LIN {X 0,Y 270.125,Z 311.646,A -85,B 0,C 180,E1 -17954.625,E2 -17954.625} C_VEL
LIN {X 0,Y 270.147,Z 311.642,A -85,B 0,C 180,E1 -17957.437,E2 -17957.437} C_VEL
LIN {X 0,Y 270.147,Z 311.617,A -85,B 0,C 180,E1 -17961.364,E2 -17961.364} C_VEL
LIN {X 0,Y 270.193,Z 311.638,A -85,B 0,C 180,E1 -17965.093,E2 -17965.093} C_VEL
LIN {X 0,Y 270.18,Z 311.636,A -85,B 0,C 180,E1 -17969.136,E2 -17969.136} C_VEL
LIN {X 0,Y 270.194,Z 311.636,A -85,B 0,C 180,E1 -17972.172,E2 -17972.172} C_VEL
LIN {X 0,Y 270.176,Z 311.639,A -85,B 0,C 180,E1 -17975.564,E2 -17975.564} C_VEL
LIN {X 0,Y 270.213,Z 311.635,A -85,B 0,C 180,E1 -17980.238,E2 -17980.238} C_VEL
LIN {X 0,Y 270.332,Z 311.614,A -85,B 0,C 180,E1 -17984.931,E2 -17984.931} C_VEL
LIN {X 0,Y 270.379,Z 311.614,A -85,B 0,C 180,E1 -17989.516,E2 -17989.516} C_VEL
LIN {X 0,Y 270.555,Z 311.591,A -85,B 0,C 180,E1 -17992.537,E2 -17992.537} C_VEL
LIN {X 0,Y 270.504,Z 311.592,A -85,B 0,C 180,E1 -17993.297,E2 -17993.297} C_VEL
LIN {X 0,Y 269.829,Z 311.675,A -85,B 0,C 180,E1 -17994.539,E2 -17994.539} C_VEL
LIN {X 0,Y 267.047,Z 312.024,A -85,B 0,C 180,E1 -17996.567,E2 -17996.567} C_VEL
LIN {X 0,Y 264.728,Z 312.32,A -85,B 0,C 180,E1 -17998.216,E2 -17998.216} C_VEL
LIN {X 0,Y 263.773,Z 312.44,A -85,B 0,C 180,E1 -17999.491,E2 -17999.491} C_VEL
LIN {X 0,Y 263.715,Z 312.449,A -85,B 0,C 180,E1 -17999.923,E2 -17999.923} C_VEL
LIN {X 0,Y 263.723,Z 312.446,A -85,B 0,C 180,E1 -18001.527,E2 -18001.527} C_VEL
LIN {X 0,Y 263.507,Z 312.47,A -85,B 0,C 180,E1 -18007.663,E2 -18007.663} C_VEL
LIN {X 0,Y 263.322,Z 312.493,A -85,B 0,C 180,E1 -18010.768,E2 -18010.768} C_VEL
LIN {X 0,Y 263.281,Z 312.494,A -85,B 0,C 180,E1 -18015.482,E2 -18015.482} C_VEL
LIN {X 0,Y 263.201,Z 312.505,A -85,B 0,C 180,E1 -18020.311,E2 -18020.311} C_VEL
LIN {X 0,Y 263.12,Z 312.522,A -85,B 0,C 180,E1 -18025.3,E2 -18025.3} C_VEL
LIN {X 0,Y 263.123,Z 312.516,A -85,B 0,C 180,E1 -18028.736,E2 -18028.736} C_VEL
LIN {X 0,Y 263.123,Z 312.52,A -85,B 0,C 180,E1 -18032.289,E2 -18032.289} C_VEL
LIN {X 0,Y 263.167,Z 312.498,A -85,B 0,C 180,E1 -18036.76,E2 -18036.76} C_VEL
LIN {X 0,Y 263.086,Z 312.497,A -85,B 0,C 180,E1 -18039.876,E2 -18039.876} C_VEL
LIN {X 0,Y 263.072,Z 312.527,A -85,B 0,C 180,E1 -18043.995,E2 -18043.995} C_VEL
LIN {X 0,Y 263.075,Z 312.505,A -85,B 0,C 180,E1 -18048.418,E2 -18048.418} C_VEL
LIN {X 0,Y 263.154,Z 312.517,A -85,B 0,C 180,E1 -18052.103,E2 -18052.103} C_VEL
LIN {X 0,Y 263.149,Z 312.509,A -85,B 0,C 180,E1 -18055.886,E2 -18055.886} C_VEL
LIN {X 0,Y 263.23,Z 312.632,A -85,B 0,C 180,E1 -18060.868,E2 -18060.868} C_VEL
LIN {X 0,Y 264.919,Z 321.271,A -85,B 0,C 180,E1 -18064.884,E2 -18064.884} C_VEL
LIN {X 0,Y 265.415,Z 323.944,A -85,B 0,C 180,E1 -18065.918,E2 -18065.918} C_VEL
LIN {X 0,Y 267.914,Z 331.705,A -85,B 0,C 180,E1 -18066.43,E2 -18066.43} C_VEL
LIN {X 0,Y 271.617,Z 351.669,A -85,B 0,C 180,E1 -18067.333,E2 -18067.333} C_VEL
LIN {X 0,Y 272.723,Z 359.199,A -85,B 0,C 180,E1 -18067.64,E2 -18067.64} C_VEL
LIN {X 0,Y 271.741,Z 400.099,A -85,B 0,C 180,E1 -18068.742,E2 -18068.742} C_VEL
LIN {X 0,Y 271.18,Z 409.643,A -85,B 0,C 180,E1 -18069.18,E2 -18069.18} C_VEL
LIN {X 0,Y 270.251,Z 420.876,A -85,B 0,C 180,E1 -18069.958,E2 -18069.958} C_VEL
LIN {X 0,Y 269.136,Z 430.854,A -85,B 0,C 180,E1 -18070.949,E2 -18070.949} C_VEL
LIN {X 0,Y 267.985,Z 439.41,A -85,B 0,C 180,E1 -18072.053,E2 -18072.053} C_VEL
LIN {X 0,Y 266.707,Z 447.46,A -85,B 0,C 180,E1 -18073.348,E2 -18073.348} C_VEL
LIN {X 0,Y 265.578,Z 454.108,A -85,B 0,C 180,E1 -18074.655,E2 -18074.655} C_VEL
LIN {X 0,Y 264.538,Z 460.419,A -85,B 0,C 180,E1 -18076.167,E2 -18076.167} C_VEL
LIN {X 0,Y 263.574,Z 465.66,A -85,B 0,C 180,E1 -18077.684,E2 -18077.684} C_VEL
LIN {X 0,Y 262.803,Z 470.03,A -85,B 0,C 180,E1 -18079.211,E2 -18079.211} C_VEL
LIN {X 0,Y 261.974,Z 475.182,A -85,B 0,C 180,E1 -18081.515,E2 -18081.515} C_VEL
LIN {X 0,Y 261.437,Z 478.962,A -85,B 0,C 180,E1 -18083.827,E2 -18083.827} C_VEL
LIN {X 0,Y 261.212,Z 480.697,A -85,B 0,C 180,E1 -18085.37,E2 -18085.37} C_VEL
LIN {X 0,Y 261.123,Z 481.938,A -85,B 0,C 180,E1 -18086.914,E2 -18086.914} C_VEL
LIN {X 0,Y 261.054,Z 482.709,A -85,B 0,C 180,E1 -18088.457,E2 -18088.457} C_VEL
LIN {X 0,Y 261.035,Z 483,A -85,B 0,C 180,E1 -18090,E2 -18090} C_VEL
LIN {X 0,Y 261.054,Z 482.702,A -85,B 0,C 180,E1 -18091.543,E2 -18091.543} C_VEL
LIN {X 0,Y 261.123,Z 481.917,A -85,B 0,C 180,E1 -18093.086,E2 -18093.086} C_VEL
LIN {X 0,Y 261.316,Z 479.565,A -85,B 0,C 180,E1 -18095.676,E2 -18095.676} C_VEL
LIN {X 0,Y 261.761,Z 476.593,A -85,B 0,C 180,E1 -18097.715,E2 -18097.715} C_VEL
LIN {X 0,Y 262.486,Z 471.858,A -85,B 0,C 180,E1 -18100.022,E2 -18100.022} C_VEL
LIN {X 0,Y 263.339,Z 466.727,A -85,B 0,C 180,E1 -18101.936,E2 -18101.936} C_VEL
LIN {X 0,Y 264.266,Z 461.711,A -85,B 0,C 180,E1 -18103.456,E2 -18103.456} C_VEL
LIN {X 0,Y 265.325,Z 455.667,A -85,B 0,C 180,E1 -18104.967,E2 -18104.967} C_VEL
LIN {X 0,Y 266.567,Z 448.31,A -85,B 0,C 180,E1 -18106.464,E2 -18106.464} C_VEL
LIN {X 0,Y 267.808,Z 440.428,A -85,B 0,C 180,E1 -18107.762,E2 -18107.762} C_VEL
LIN {X 0,Y 268.955,Z 432.094,A -85,B 0,C 180,E1 -18108.866,E2 -18108.866} C_VEL
LIN {X 0,Y 270.138,Z 421.49,A -85,B 0,C 180,E1 -18109.96,E2 -18109.96} C_VEL
LIN {X 0,Y 271.066,Z 410.29,A -85,B 0,C 180,E1 -18110.756,E2 -18110.756} C_VEL
LIN {X 0,Y 271.665,Z 400.812,A -85,B 0,C 180,E1 -18111.202,E2 -18111.202} C_VEL
LIN {X 0,Y 272.674,Z 360.484,A -85,B 0,C 180,E1 -18112.293,E2 -18112.293} C_VEL
LIN {X 0,Y 271.694,Z 352.525,A -85,B 0,C 180,E1 -18112.601,E2 -18112.601} C_VEL
LIN {X 0,Y 268.016,Z 332.206,A -85,B 0,C 180,E1 -18113.509,E2 -18113.509} C_VEL
LIN {X 0,Y 265.417,Z 324.066,A -85,B 0,C 180,E1 -18114.026,E2 -18114.026} C_VEL
LIN {X 0,Y 265.197,Z 322.835,A -85,B 0,C 180,E1 -18114.388,E2 -18114.388} C_VEL
LIN {X 0,Y 263.296,Z 312.887,A -85,B 0,C 180,E1 -18118.933,E2 -18118.933} C_VEL
LIN {X 0,Y 263.185,Z 312.512,A -85,B 0,C 180,E1 -18119.604,E2 -18119.604} C_VEL
LIN {X 0,Y 263.149,Z 312.509,A -85,B 0,C 180,E1 -18124.114,E2 -18124.114} C_VEL
LIN {X 0,Y 263.154,Z 312.517,A -85,B 0,C 180,E1 -18127.897,E2 -18127.897} C_VEL
LIN {X 0,Y 263.075,Z 312.507,A -85,B 0,C 180,E1 -18131.902,E2 -18131.902} C_VEL
LIN {X 0,Y 263.074,Z 312.527,A -85,B 0,C 180,E1 -18136.161,E2 -18136.161} C_VEL
LIN {X 0,Y 263.108,Z 312.49,A -85,B 0,C 180,E1 -18140.77,E2 -18140.77} C_VEL
LIN {X 0,Y 263.15,Z 312.508,A -85,B 0,C 180,E1 -18144.016,E2 -18144.016} C_VEL
LIN {X 0,Y 263.123,Z 312.52,A -85,B 0,C 180,E1 -18147.711,E2 -18147.711} C_VEL
LIN {X 0,Y 263.139,Z 312.514,A -85,B 0,C 180,E1 -18151.806,E2 -18151.806} C_VEL
LIN {X 0,Y 263.108,Z 312.517,A -85,B 0,C 180,E1 -18156.38,E2 -18156.38} C_VEL
LIN {X 0,Y 263.201,Z 312.506,A -85,B 0,C 180,E1 -18159.689,E2 -18159.689} C_VEL
LIN {X 0,Y 263.281,Z 312.494,A -85,B 0,C 180,E1 -18164.518,E2 -18164.518} C_VEL
LIN {X 0,Y 263.323,Z 312.493,A -85,B 0,C 180,E1 -18169.232,E2 -18169.232} C_VEL
LIN {X 0,Y 263.519,Z 312.469,A -85,B 0,C 180,E1 -18172.337,E2 -18172.337} C_VEL
LIN {X 0,Y 263.725,Z 312.446,A -85,B 0,C 180,E1 -18178.473,E2 -18178.473} C_VEL
LIN {X 0,Y 263.723,Z 312.446,A -85,B 0,C 180,E1 -18181.527,E2 -18181.527} C_VEL
LIN {X 0,Y 263.507,Z 312.47,A -85,B 0,C 180,E1 -18187.664,E2 -18187.664} C_VEL
LIN {X 0,Y 263.322,Z 312.493,A -85,B 0,C 180,E1 -18190.768,E2 -18190.768} C_VEL
LIN {X 0,Y 263.282,Z 312.493,A -85,B 0,C 180,E1 -18195.482,E2 -18195.482} C_VEL
LIN {X 0,Y 263.201,Z 312.506,A -85,B 0,C 180,E1 -18200.312,E2 -18200.312} C_VEL
LIN {X 0,Y 263.12,Z 312.522,A -85,B 0,C 180,E1 -18205.301,E2 -18205.301} C_VEL
LIN {X 0,Y 263.124,Z 312.517,A -85,B 0,C 180,E1 -18208.736,E2 -18208.736} C_VEL
LIN {X 0,Y 263.123,Z 312.519,A -85,B 0,C 180,E1 -18212.29,E2 -18212.29} C_VEL
LIN {X 0,Y 263.168,Z 312.499,A -85,B 0,C 180,E1 -18216.761,E2 -18216.761} C_VEL
LIN {X 0,Y 263.087,Z 312.495,A -85,B 0,C 180,E1 -18219.876,E2 -18219.876} C_VEL
LIN {X 0,Y 263.073,Z 312.527,A -85,B 0,C 180,E1 -18223.995,E2 -18223.995} C_VEL
LIN {X 0,Y 263.076,Z 312.506,A -85,B 0,C 180,E1 -18228.419,E2 -18228.419} C_VEL
LIN {X 0,Y 263.155,Z 312.517,A -85,B 0,C 180,E1 -18232.103,E2 -18232.103} C_VEL
LIN {X 0,Y 263.15,Z 312.508,A -85,B 0,C 180,E1 -18235.886,E2 -18235.886} C_VEL
LIN {X 0,Y 263.128,Z 312.52,A -85,B 0,C 180,E1 -18240.389,E2 -18240.389} C_VEL
LIN {X 0,Y 263.199,Z 312.797,A -85,B 0,C 180,E1 -18241.055,E2 -18241.055} C_VEL
LIN {X 0,Y 264.895,Z 321.076,A -85,B 0,C 180,E1 -18244.882,E2 -18244.882} C_VEL
LIN {X 0,Y 265.369,Z 323.811,A -85,B 0,C 180,E1 -18245.98,E2 -18245.98} C_VEL
LIN {X 0,Y 267.627,Z 330.782,A -85,B 0,C 180,E1 -18246.459,E2 -18246.459} C_VEL
LIN {X 0,Y 270.957,Z 347.701,A -85,B 0,C 180,E1 -18247.243,E2 -18247.243} C_VEL
LIN {X 0,Y 272.661,Z 359.429,A -85,B 0,C 180,E1 -18247.721,E2 -18247.721} C_VEL
LIN {X 0,Y 271.615,Z 400.572,A -85,B 0,C 180,E1 -18248.829,E2 -18248.829} C_VEL
LIN {X 0,Y 271.081,Z 410.526,A -85,B 0,C 180,E1 -18249.304,E2 -18249.304} C_VEL
LIN {X 0,Y 270.219,Z 421.026,A -85,B 0,C 180,E1 -18250.048,E2 -18250.048} C_VEL
LIN {X 0,Y 269.026,Z 431.752,A -85,B 0,C 180,E1 -18251.139,E2 -18251.139} C_VEL
LIN {X 0,Y 267.806,Z 440.147,A -85,B 0,C 180,E1 -18252.238,E2 -18252.238} C_VEL
LIN {X 0,Y 266.603,Z 448.077,A -85,B 0,C 180,E1 -18253.538,E2 -18253.538} C_VEL
LIN {X 0,Y 265.355,Z 455.472,A -85,B 0,C 180,E1 -18255.035,E2 -18255.035} C_VEL
LIN {X 0,Y 264.049,Z 462.964,A -85,B 0,C 180,E1 -18256.925,E2 -18256.925} C_VEL
LIN {X 0,Y 262.854,Z 469.835,A -85,B 0,C 180,E1 -18259.213,E2 -18259.213} C_VEL
LIN {X 0,Y 261.981,Z 475.029,A -85,B 0,C 180,E1 -18261.516,E2 -18261.516} C_VEL
LIN {X 0,Y 261.562,Z 477.695,A -85,B 0,C 180,E1 -18263.055,E2 -18263.055} C_VEL
LIN {X 0,Y 261.319,Z 479.512,A -85,B 0,C 180,E1 -18264.321,E2 -18264.321} C_VEL
LIN {X 0,Y 261.126,Z 481.889,A -85,B 0,C 180,E1 -18266.914,E2 -18266.914} C_VEL
LIN {X 0,Y 261.055,Z 482.692,A -85,B 0,C 180,E1 -18268.457,E2 -18268.457} C_VEL
LIN {X 0,Y 261.036,Z 482.998,A -85,B 0,C 180,E1 -18270,E2 -18270} C_VEL
LIN {X 0,Y 261.051,Z 482.718,A -85,B 0,C 180,E1 -18271.543,E2 -18271.543} C_VEL
LIN {X 0,Y 261.096,Z 481.966,A -85,B 0,C 180,E1 -18273.086,E2 -18273.086} C_VEL
LIN {X 0,Y 261.306,Z 479.677,A -85,B 0,C 180,E1 -18275.648,E2 -18275.648} C_VEL
LIN {X 0,Y 261.762,Z 476.721,A -85,B 0,C 180,E1 -18277.715,E2 -18277.715} C_VEL
LIN {X 0,Y 262.467,Z 472.051,A -85,B 0,C 180,E1 -18280.023,E2 -18280.023} C_VEL
LIN {X 0,Y 263.339,Z 466.967,A -85,B 0,C 180,E1 -18281.936,E2 -18281.936} C_VEL
LIN {X 0,Y 264.262,Z 462,A -85,B 0,C 180,E1 -18283.456,E2 -18283.456} C_VEL
LIN {X 0,Y 265.278,Z 456.007,A -85,B 0,C 180,E1 -18284.969,E2 -18284.969} C_VEL
LIN {X 0,Y 266.494,Z 448.713,A -85,B 0,C 180,E1 -18286.469,E2 -18286.469} C_VEL
LIN {X 0,Y 267.784,Z 440.919,A -85,B 0,C 180,E1 -18287.764,E2 -18287.764} C_VEL
LIN {X 0,Y 268.969,Z 432.696,A -85,B 0,C 180,E1 -18288.865,E2 -18288.865} C_VEL
LIN {X 0,Y 269.934,Z 424.107,A -85,B 0,C 180,E1 -18289.783,E2 -18289.783} C_VEL
LIN {X 0,Y 270.869,Z 414.122,A -85,B 0,C 180,E1 -18290.594,E2 -18290.594} C_VEL
LIN {X 0,Y 271.632,Z 402.078,A -85,B 0,C 180,E1 -18291.236,E2 -18291.236} C_VEL
LIN {X 0,Y 272.157,Z 381.681,A -85,B 0,C 180,E1 -18291.827,E2 -18291.827} C_VEL
LIN {X 0,Y 272.664,Z 358.428,A -85,B 0,C 180,E1 -18292.432,E2 -18292.432} C_VEL
LIN {X 0,Y 268.973,Z 336.642,A -85,B 0,C 180,E1 -18293.375,E2 -18293.375} C_VEL
LIN {X 0,Y 267.008,Z 328.675,A -85,B 0,C 180,E1 -18293.787,E2 -18293.787} C_VEL
LIN {X 0,Y 265.366,Z 323.842,A -85,B 0,C 180,E1 -18294.144,E2 -18294.144} C_VEL
LIN {X 0,Y 264.499,Z 319.23,A -85,B 0,C 180,E1 -18296.086,E2 -18296.086} C_VEL
LIN {X 0,Y 263.211,Z 312.616,A -85,B 0,C 180,E1 -18299.217,E2 -18299.217} C_VEL
LIN {X 0,Y 263.15,Z 312.509,A -85,B 0,C 180,E1 -18304.114,E2 -18304.114} C_VEL
LIN {X 0,Y 263.155,Z 312.517,A -85,B 0,C 180,E1 -18307.897,E2 -18307.897} C_VEL
LIN {X 0,Y 263.076,Z 312.506,A -85,B 0,C 180,E1 -18311.901,E2 -18311.901} C_VEL
LIN {X 0,Y 263.075,Z 312.527,A -85,B 0,C 180,E1 -18316.16,E2 -18316.16} C_VEL
LIN {X 0,Y 263.068,Z 312.499,A -85,B 0,C 180,E1 -18320.12,E2 -18320.12} C_VEL
LIN {X 0,Y 263.149,Z 312.508,A -85,B 0,C 180,E1 -18324.016,E2 -18324.016} C_VEL
LIN {X 0,Y 263.124,Z 312.52,A -85,B 0,C 180,E1 -18327.71,E2 -18327.71} C_VEL
LIN {X 0,Y 263.14,Z 312.514,A -85,B 0,C 180,E1 -18331.806,E2 -18331.806} C_VEL
LIN {X 0,Y 263.109,Z 312.517,A -85,B 0,C 180,E1 -18336.38,E2 -18336.38} C_VEL
LIN {X 0,Y 263.201,Z 312.505,A -85,B 0,C 180,E1 -18339.688,E2 -18339.688} C_VEL
LIN {X 0,Y 263.282,Z 312.494,A -85,B 0,C 180,E1 -18344.518,E2 -18344.518} C_VEL
LIN {X 0,Y 263.323,Z 312.493,A -85,B 0,C 180,E1 -18349.232,E2 -18349.232} C_VEL
LIN {X 0,Y 263.519,Z 312.469,A -85,B 0,C 180,E1 -18352.337,E2 -18352.337} C_VEL
LIN {X 0,Y 263.725,Z 312.446,A -85,B 0,C 180,E1 -18358.473,E2 -18358.473} C_VEL
LIN {X 0,Y 263.715,Z 312.449,A -85,B 0,C 180,E1 -18359.923,E2 -18359.923} C_VEL
LIN {X 0,Y 263.429,Z 312.49,A -85,B 0,C 180,E1 -18360.773,E2 -18360.773} C_VEL
LIN {X 0,Y 262.076,Z 312.661,A -85,B 0,C 180,E1 -18362.026,E2 -18362.026} C_VEL
LIN {X 0,Y 257.623,Z 313.202,A -85,B 0,C 180,E1 -18364.943,E2 -18364.943} C_VEL
LIN {X 0,Y 256.522,Z 313.334,A -85,B 0,C 180,E1 -18366.25,E2 -18366.25} C_VEL
LIN {X 0,Y 256.426,Z 313.346,A -85,B 0,C 180,E1 -18366.694,E2 -18366.694} C_VEL
LIN {X 0,Y 256.393,Z 313.36,A -85,B 0,C 180,E1 -18369.466,E2 -18369.466} C_VEL
LIN {X 0,Y 256.193,Z 313.371,A -85,B 0,C 180,E1 -18374.294,E2 -18374.294} C_VEL
LIN {X 0,Y 256.141,Z 313.392,A -85,B 0,C 180,E1 -18377.567,E2 -18377.567} C_VEL
LIN {X 0,Y 256.113,Z 313.386,A -85,B 0,C 180,E1 -18381.097,E2 -18381.097} C_VEL
LIN {X 0,Y 256.079,Z 313.397,A -85,B 0,C 180,E1 -18385.089,E2 -18385.089} C_VEL
LIN {X 0,Y 256.081,Z 313.393,A -85,B 0,C 180,E1 -18388.574,E2 -18388.574} C_VEL
LIN {X 0,Y 256.069,Z 313.4,A -85,B 0,C 180,E1 -18391.702,E2 -18391.702} C_VEL
LIN {X 0,Y 256.073,Z 313.393,A -85,B 0,C 180,E1 -18395.194,E2 -18395.194} C_VEL
LIN {X 0,Y 256.059,Z 313.366,A -85,B 0,C 180,E1 -18399.144,E2 -18399.144} C_VEL
LIN {X 0,Y 256.018,Z 313.408,A -85,B 0,C 180,E1 -18403.336,E2 -18403.336} C_VEL
LIN {X 0,Y 256.029,Z 313.383,A -85,B 0,C 180,E1 -18407.829,E2 -18407.829} C_VEL
LIN {X 0,Y 256.063,Z 313.394,A -85,B 0,C 180,E1 -18410.857,E2 -18410.857} C_VEL
LIN {X 0,Y 256.123,Z 313.392,A -85,B 0,C 180,E1 -18412.867,E2 -18412.867} C_VEL
LIN {X 0,Y 256.064,Z 313.399,A -85,B 0,C 180,E1 -18416.708,E2 -18416.708} C_VEL
LIN {X 0,Y 256.152,Z 313.535,A -85,B 0,C 180,E1 -18420.406,E2 -18420.406} C_VEL
LIN {X 0,Y 257.315,Z 319.321,A -85,B 0,C 180,E1 -18423.215,E2 -18423.215} C_VEL
LIN {X 0,Y 258.17,Z 323.787,A -85,B 0,C 180,E1 -18425.174,E2 -18425.174} C_VEL
LIN {X 0,Y 260.374,Z 329.726,A -85,B 0,C 180,E1 -18425.645,E2 -18425.645} C_VEL
LIN {X 0,Y 262.419,Z 337.483,A -85,B 0,C 180,E1 -18426.075,E2 -18426.075} C_VEL
LIN {X 0,Y 265.87,Z 357.852,A -85,B 0,C 180,E1 -18426.992,E2 -18426.992} C_VEL
LIN {X 0,Y 266.136,Z 361.772,A -85,B 0,C 180,E1 -18427.129,E2 -18427.129} C_VEL
LIN {X 0,Y 265.164,Z 399.495,A -85,B 0,C 180,E1 -18428.163,E2 -18428.163} C_VEL
LIN {X 0,Y 264.608,Z 409.016,A -85,B 0,C 180,E1 -18428.599,E2 -18428.599} C_VEL
LIN {X 0,Y 263.738,Z 418.936,A -85,B 0,C 180,E1 -18429.275,E2 -18429.275} C_VEL
LIN {X 0,Y 262.724,Z 429.274,A -85,B 0,C 180,E1 -18430.262,E2 -18430.262} C_VEL
LIN {X 0,Y 261.252,Z 439.413,A -85,B 0,C 180,E1 -18431.574,E2 -18431.574} C_VEL
LIN {X 0,Y 259.917,Z 447.463,A -85,B 0,C 180,E1 -18432.9,E2 -18432.9} C_VEL
LIN {X 0,Y 258.734,Z 454.111,A -85,B 0,C 180,E1 -18434.239,E2 -18434.239} C_VEL
LIN {X 0,Y 257.631,Z 460.421,A -85,B 0,C 180,E1 -18435.788,E2 -18435.788} C_VEL
LIN {X 0,Y 256.622,Z 465.662,A -85,B 0,C 180,E1 -18437.345,E2 -18437.345} C_VEL
LIN {X 0,Y 255.823,Z 470.031,A -85,B 0,C 180,E1 -18438.913,E2 -18438.913} C_VEL
LIN {X 0,Y 254.936,Z 475.183,A -85,B 0,C 180,E1 -18441.279,E2 -18441.279} C_VEL
LIN {X 0,Y 254.373,Z 478.963,A -85,B 0,C 180,E1 -18443.655,E2 -18443.655} C_VEL
LIN {X 0,Y 254.137,Z 480.698,A -85,B 0,C 180,E1 -18445.241,E2 -18445.241} C_VEL
LIN {X 0,Y 254.026,Z 481.939,A -85,B 0,C 180,E1 -18446.828,E2 -18446.828} C_VEL
LIN {X 0,Y 253.966,Z 482.709,A -85,B 0,C 180,E1 -18448.414,E2 -18448.414} C_VEL
LIN {X 0,Y 253.945,Z 483,A -85,B 0,C 180,E1 -18450,E2 -18450} C_VEL
LIN {X 0,Y 253.966,Z 482.702,A -85,B 0,C 180,E1 -18451.586,E2 -18451.586} C_VEL
LIN {X 0,Y 254.025,Z 481.917,A -85,B 0,C 180,E1 -18453.172,E2 -18453.172} C_VEL
LIN {X 0,Y 254.204,Z 479.844,A -85,B 0,C 180,E1 -18455.562,E2 -18455.562} C_VEL
LIN {X 0,Y 254.719,Z 476.592,A -85,B 0,C 180,E1 -18457.929,E2 -18457.929} C_VEL
LIN {X 0,Y 255.475,Z 471.856,A -85,B 0,C 180,E1 -18460.3,E2 -18460.3} C_VEL
LIN {X 0,Y 256.393,Z 466.725,A -85,B 0,C 180,E1 -18462.265,E2 -18462.265} C_VEL
LIN {X 0,Y 257.37,Z 461.709,A -85,B 0,C 180,E1 -18463.823,E2 -18463.823} C_VEL
LIN {X 0,Y 258.447,Z 455.664,A -85,B 0,C 180,E1 -18465.375,E2 -18465.375} C_VEL
LIN {X 0,Y 259.767,Z 448.307,A -85,B 0,C 180,E1 -18466.908,E2 -18466.908} C_VEL
LIN {X 0,Y 261.064,Z 440.424,A -85,B 0,C 180,E1 -18468.237,E2 -18468.237} C_VEL
LIN {X 0,Y 262.261,Z 432.089,A -85,B 0,C 180,E1 -18469.367,E2 -18469.367} C_VEL
LIN {X 0,Y 263.469,Z 421.59,A -85,B 0,C 180,E1 -18470.477,E2 -18470.477} C_VEL
LIN {X 0,Y 264.441,Z 410.455,A -85,B 0,C 180,E1 -18471.29,E2 -18471.29} C_VEL
LIN {X 0,Y 265.071,Z 400.912,A -85,B 0,C 180,E1 -18471.752,E2 -18471.752} C_VEL
LIN {X 0,Y 266.033,Z 364.759,A -85,B 0,C 180,E1 -18472.758,E2 -18472.758} C_VEL
LIN {X 0,Y 265.954,Z 358.587,A -85,B 0,C 180,E1 -18472.942,E2 -18472.942} C_VEL
LIN {X 0,Y 262.097,Z 336.182,A -85,B 0,C 180,E1 -18473.955,E2 -18473.955} C_VEL
LIN {X 0,Y 260.124,Z 329.253,A -85,B 0,C 180,E1 -18474.354,E2 -18474.354} C_VEL
LIN {X 0,Y 258.2,Z 323.811,A -85,B 0,C 180,E1 -18474.777,E2 -18474.777} C_VEL
LIN {X 0,Y 256.717,Z 316.204,A -85,B 0,C 180,E1 -18478.222,E2 -18478.222} C_VEL
LIN {X 0,Y 256.155,Z 313.494,A -85,B 0,C 180,E1 -18479.594,E2 -18479.594} C_VEL
LIN {X 0,Y 256.102,Z 313.383,A -85,B 0,C 180,E1 -18484.587,E2 -18484.587} C_VEL
LIN {X 0,Y 256.107,Z 313.396,A -85,B 0,C 180,E1 -18487.269,E2 -18487.269} C_VEL
LIN {X 0,Y 256.013,Z 313.383,A -85,B 0,C 180,E1 -18491.21,E2 -18491.21} C_VEL
LIN {X 0,Y 256.013,Z 313.408,A -85,B 0,C 180,E1 -18495.539,E2 -18495.539} C_VEL
LIN {X 0,Y 256.013,Z 313.387,A -85,B 0,C 180,E1 -18498.789,E2 -18498.789} C_VEL
LIN {X 0,Y 256.097,Z 313.374,A -85,B 0,C 180,E1 -18502.862,E2 -18502.862} C_VEL
LIN {X 0,Y 256.061,Z 313.403,A -85,B 0,C 180,E1 -18506.706,E2 -18506.706} C_VEL
LIN {X 0,Y 256.046,Z 313.392,A -85,B 0,C 180,E1 -18510.392,E2 -18510.392} C_VEL
LIN {X 0,Y 256.068,Z 313.4,A -85,B 0,C 180,E1 -18513.952,E2 -18513.952} C_VEL
LIN {X 0,Y 256.05,Z 313.388,A -85,B 0,C 180,E1 -18517.402,E2 -18517.402} C_VEL
LIN {X 0,Y 256.1,Z 313.397,A -85,B 0,C 180,E1 -18520.773,E2 -18520.773} C_VEL
LIN {X 0,Y 256.206,Z 313.379,A -85,B 0,C 180,E1 -18524.079,E2 -18524.079} C_VEL
LIN {X 0,Y 256.267,Z 313.372,A -85,B 0,C 180,E1 -18528.932,E2 -18528.932} C_VEL
LIN {X 0,Y 256.483,Z 313.347,A -85,B 0,C 180,E1 -18532.125,E2 -18532.125} C_VEL
LIN {X 0,Y 256.441,Z 313.346,A -85,B 0,C 180,E1 -18536.858,E2 -18536.858} C_VEL
LIN {X 0,Y 256.688,Z 313.323,A -85,B 0,C 180,E1 -18538.431,E2 -18538.431} C_VEL
LIN {X 0,Y 256.686,Z 313.323,A -85,B 0,C 180,E1 -18541.569,E2 -18541.569} C_VEL
LIN {X 0,Y 256.43,Z 313.345,A -85,B 0,C 180,E1 -18546.564,E2 -18546.564} C_VEL
LIN {X 0,Y 256.393,Z 313.36,A -85,B 0,C 180,E1 -18549.466,E2 -18549.466} C_VEL
LIN {X 0,Y 256.193,Z 313.371,A -85,B 0,C 180,E1 -18554.294,E2 -18554.294} C_VEL
LIN {X 0,Y 256.141,Z 313.392,A -85,B 0,C 180,E1 -18557.567,E2 -18557.567} C_VEL
LIN {X 0,Y 256.113,Z 313.386,A -85,B 0,C 180,E1 -18561.097,E2 -18561.097} C_VEL
LIN {X 0,Y 256.079,Z 313.397,A -85,B 0,C 180,E1 -18565.089,E2 -18565.089} C_VEL
LIN {X 0,Y 256.081,Z 313.393,A -85,B 0,C 180,E1 -18568.574,E2 -18568.574} C_VEL
LIN {X 0,Y 256.07,Z 313.4,A -85,B 0,C 180,E1 -18571.702,E2 -18571.702} C_VEL
LIN {X 0,Y 256.074,Z 313.394,A -85,B 0,C 180,E1 -18575.194,E2 -18575.194} C_VEL
LIN {X 0,Y 256.06,Z 313.366,A -85,B 0,C 180,E1 -18579.144,E2 -18579.144} C_VEL
LIN {X 0,Y 256.019,Z 313.407,A -85,B 0,C 180,E1 -18583.336,E2 -18583.336} C_VEL
LIN {X 0,Y 256.03,Z 313.385,A -85,B 0,C 180,E1 -18587.83,E2 -18587.83} C_VEL
LIN {X 0,Y 256.064,Z 313.393,A -85,B 0,C 180,E1 -18590.858,E2 -18590.858} C_VEL
LIN {X 0,Y 256.124,Z 313.393,A -85,B 0,C 180,E1 -18592.867,E2 -18592.867} C_VEL
LIN {X 0,Y 256.064,Z 313.397,A -85,B 0,C 180,E1 -18596.708,E2 -18596.708} C_VEL
LIN {X 0,Y 256.117,Z 313.602,A -85,B 0,C 180,E1 -18600.535,E2 -18600.535} C_VEL
LIN {X 0,Y 257.682,Z 321.16,A -85,B 0,C 180,E1 -18604.164,E2 -18604.164} C_VEL
LIN {X 0,Y 258.213,Z 323.848,A -85,B 0,C 180,E1 -18605.275,E2 -18605.275} C_VEL
LIN {X 0,Y 261.273,Z 332.699,A -85,B 0,C 180,E1 -18605.907,E2 -18605.907} C_VEL
LIN {X 0,Y 264.171,Z 347.24,A -85,B 0,C 180,E1 -18606.611,E2 -18606.611} C_VEL
LIN {X 0,Y 266.089,Z 360.409,A -85,B 0,C 180,E1 -18607.168,E2 -18607.168} C_VEL
LIN {X 0,Y 265.047,Z 400.178,A -85,B 0,C 180,E1 -18608.262,E2 -18608.262} C_VEL
LIN {X 0,Y 264.499,Z 409.831,A -85,B 0,C 180,E1 -18608.722,E2 -18608.722} C_VEL
LIN {X 0,Y 263.549,Z 421.135,A -85,B 0,C 180,E1 -18609.53,E2 -18609.53} C_VEL
LIN {X 0,Y 262.33,Z 431.757,A -85,B 0,C 180,E1 -18610.639,E2 -18610.639} C_VEL
LIN {X 0,Y 261.053,Z 440.151,A -85,B 0,C 180,E1 -18611.762,E2 -18611.762} C_VEL
LIN {X 0,Y 259.807,Z 448.08,A -85,B 0,C 180,E1 -18613.095,E2 -18613.095} C_VEL
LIN {X 0,Y 258.5,Z 455.475,A -85,B 0,C 180,E1 -18614.629,E2 -18614.629} C_VEL
LIN {X 0,Y 257.121,Z 462.967,A -85,B 0,C 180,E1 -18616.566,E2 -18616.566} C_VEL
LIN {X 0,Y 255.859,Z 469.836,A -85,B 0,C 180,E1 -18618.915,E2 -18618.915} C_VEL
LIN {X 0,Y 254.943,Z 475.03,A -85,B 0,C 180,E1 -18621.279,E2 -18621.279} C_VEL
LIN {X 0,Y 254.514,Z 477.696,A -85,B 0,C 180,E1 -18622.862,E2 -18622.862} C_VEL
LIN {X 0,Y 254.135,Z 480.615,A -85,B 0,C 180,E1 -18625.241,E2 -18625.241} C_VEL
LIN {X 0,Y 254.028,Z 481.889,A -85,B 0,C 180,E1 -18626.828,E2 -18626.828} C_VEL
LIN {X 0,Y 253.968,Z 482.693,A -85,B 0,C 180,E1 -18628.414,E2 -18628.414} C_VEL
LIN {X 0,Y 253.946,Z 482.998,A -85,B 0,C 180,E1 -18630,E2 -18630} C_VEL
LIN {X 0,Y 253.963,Z 482.718,A -85,B 0,C 180,E1 -18631.586,E2 -18631.586} C_VEL
LIN {X 0,Y 253.999,Z 481.966,A -85,B 0,C 180,E1 -18633.172,E2 -18633.172} C_VEL
LIN {X 0,Y 254.184,Z 479.976,A -85,B 0,C 180,E1 -18635.513,E2 -18635.513} C_VEL
LIN {X 0,Y 254.719,Z 476.72,A -85,B 0,C 180,E1 -18637.929,E2 -18637.929} C_VEL
LIN {X 0,Y 255.457,Z 472.049,A -85,B 0,C 180,E1 -18640.301,E2 -18640.301} C_VEL
LIN {X 0,Y 256.394,Z 466.965,A -85,B 0,C 180,E1 -18642.265,E2 -18642.265} C_VEL
LIN {X 0,Y 257.364,Z 461.998,A -85,B 0,C 180,E1 -18643.824,E2 -18643.824} C_VEL
LIN {X 0,Y 258.4,Z 456.004,A -85,B 0,C 180,E1 -18645.377,E2 -18645.377} C_VEL
LIN {X 0,Y 259.708,Z 448.71,A -85,B 0,C 180,E1 -18646.912,E2 -18646.912} C_VEL
LIN {X 0,Y 261.033,Z 440.915,A -85,B 0,C 180,E1 -18648.239,E2 -18648.239} C_VEL
LIN {X 0,Y 262.27,Z 432.691,A -85,B 0,C 180,E1 -18649.366,E2 -18649.366} C_VEL
LIN {X 0,Y 263.28,Z 424.101,A -85,B 0,C 180,E1 -18650.305,E2 -18650.305} C_VEL
LIN {X 0,Y 264.263,Z 413.686,A -85,B 0,C 180,E1 -18651.169,E2 -18651.169} C_VEL
LIN {X 0,Y 265.029,Z 402.061,A -85,B 0,C 180,E1 -18651.792,E2 -18651.792} C_VEL
LIN {X 0,Y 265.56,Z 382.385,A -85,B 0,C 180,E1 -18652.377,E2 -18652.377} C_VEL
LIN {X 0,Y 266.16,Z 359.776,A -85,B 0,C 180,E1 -18652.971,E2 -18652.971} C_VEL
LIN {X 0,Y 262.508,Z 337.898,A -85,B 0,C 180,E1 -18653.949,E2 -18653.949} C_VEL
LIN {X 0,Y 260.616,Z 330.58,A -85,B 0,C 180,E1 -18654.351,E2 -18654.351} C_VEL
LIN {X 0,Y 258.291,Z 324.185,A -85,B 0,C 180,E1 -18654.814,E2 -18654.814} C_VEL
LIN {X 0,Y 258.058,Z 323.085,A -85,B 0,C 180,E1 -18655.102,E2 -18655.102} C_VEL
LIN {X 0,Y 256.518,Z 315.297,A -85,B 0,C 180,E1 -18658.75,E2 -18658.75} C_VEL
LIN {X 0,Y 256.14,Z 313.488,A -85,B 0,C 180,E1 -18659.709,E2 -18659.709} C_VEL
LIN {X 0,Y 256.103,Z 313.383,A -85,B 0,C 180,E1 -18664.587,E2 -18664.587} C_VEL
LIN {X 0,Y 256.108,Z 313.395,A -85,B 0,C 180,E1 -18667.268,E2 -18667.268} C_VEL
LIN {X 0,Y 256.014,Z 313.383,A -85,B 0,C 180,E1 -18671.21,E2 -18671.21} C_VEL
LIN {X 0,Y 256.014,Z 313.408,A -85,B 0,C 180,E1 -18675.539,E2 -18675.539} C_VEL
LIN {X 0,Y 256.005,Z 313.39,A -85,B 0,C 180,E1 -18678.787,E2 -18678.787} C_VEL
LIN {X 0,Y 256.095,Z 313.373,A -85,B 0,C 180,E1 -18682.861,E2 -18682.861} C_VEL
LIN {X 0,Y 256.062,Z 313.402,A -85,B 0,C 180,E1 -18686.706,E2 -18686.706} C_VEL
LIN {X 0,Y 256.047,Z 313.392,A -85,B 0,C 180,E1 -18690.392,E2 -18690.392} C_VEL
LIN {X 0,Y 256.068,Z 313.399,A -85,B 0,C 180,E1 -18693.951,E2 -18693.951} C_VEL
LIN {X 0,Y 256.051,Z 313.389,A -85,B 0,C 180,E1 -18697.402,E2 -18697.402} C_VEL
LIN {X 0,Y 256.1,Z 313.397,A -85,B 0,C 180,E1 -18700.773,E2 -18700.773} C_VEL
LIN {X 0,Y 256.207,Z 313.379,A -85,B 0,C 180,E1 -18704.079,E2 -18704.079} C_VEL
LIN {X 0,Y 256.267,Z 313.372,A -85,B 0,C 180,E1 -18708.932,E2 -18708.932} C_VEL
LIN {X 0,Y 256.483,Z 313.347,A -85,B 0,C 180,E1 -18712.125,E2 -18712.125} C_VEL
LIN {X 0,Y 256.441,Z 313.346,A -85,B 0,C 180,E1 -18716.858,E2 -18716.858} C_VEL
LIN {X 0,Y 256.688,Z 313.323,A -85,B 0,C 180,E1 -18718.431,E2 -18718.431} C_VEL
LIN {X 0,Y 256.686,Z 313.323,A -85,B 0,C 180,E1 -18721.569,E2 -18721.569} C_VEL
LIN {X 0,Y 256.426,Z 313.346,A -85,B 0,C 180,E1 -18726.694,E2 -18726.694} C_VEL
LIN {X 0,Y 255.723,Z 313.443,A -85,B 0,C 180,E1 -18728.004,E2 -18728.004} C_VEL
LIN {X 0,Y 252.788,Z 313.807,A -85,B 0,C 180,E1 -18730.137,E2 -18730.137} C_VEL
LIN {X 0,Y 250.297,Z 314.11,A -85,B 0,C 180,E1 -18731.873,E2 -18731.873} C_VEL
LIN {X 0,Y 249.218,Z 314.239,A -85,B 0,C 180,E1 -18733.221,E2 -18733.221} C_VEL
LIN {X 0,Y 249.124,Z 314.249,A -85,B 0,C 180,E1 -18733.679,E2 -18733.679} C_VEL
LIN {X 0,Y 249.145,Z 314.259,A -85,B 0,C 180,E1 -18736.45,E2 -18736.45} C_VEL
LIN {X 0,Y 249.037,Z 314.263,A -85,B 0,C 180,E1 -18741.522,E2 -18741.522} C_VEL
LIN {X 0,Y 249.041,Z 314.277,A -85,B 0,C 180,E1 -18745.441,E2 -18745.441} C_VEL
LIN {X 0,Y 249.028,Z 314.268,A -85,B 0,C 180,E1 -18748.973,E2 -18748.973} C_VEL
LIN {X 0,Y 249.023,Z 314.277,A -85,B 0,C 180,E1 -18752.427,E2 -18752.427} C_VEL
LIN {X 0,Y 249.006,Z 314.264,A -85,B 0,C 180,E1 -18756.349,E2 -18756.349} C_VEL
LIN {X 0,Y 248.974,Z 314.256,A -85,B 0,C 180,E1 -18760.484,E2 -18760.484} C_VEL
LIN {X 0,Y 248.958,Z 314.286,A -85,B 0,C 180,E1 -18764.889,E2 -18764.889} C_VEL
LIN {X 0,Y 248.975,Z 314.265,A -85,B 0,C 180,E1 -18767.355,E2 -18767.355} C_VEL
LIN {X 0,Y 249.037,Z 314.277,A -85,B 0,C 180,E1 -18772.202,E2 -18772.202} C_VEL
LIN {X 0,Y 249.04,Z 314.263,A -85,B 0,C 180,E1 -18775.64,E2 -18775.64} C_VEL
LIN {X 0,Y 249.101,Z 314.437,A -85,B 0,C 180,E1 -18779.918,E2 -18779.918} C_VEL
LIN {X 0,Y 250.486,Z 321.275,A -85,B 0,C 180,E1 -18783.326,E2 -18783.326} C_VEL
LIN {X 0,Y 250.966,Z 323.787,A -85,B 0,C 180,E1 -18784.41,E2 -18784.41} C_VEL
LIN {X 0,Y 253.214,Z 329.689,A -85,B 0,C 180,E1 -18784.908,E2 -18784.908} C_VEL
LIN {X 0,Y 255.725,Z 337.464,A -85,B 0,C 180,E1 -18785.407,E2 -18785.407} C_VEL
LIN {X 0,Y 259.107,Z 357.248,A -85,B 0,C 180,E1 -18786.337,E2 -18786.337} C_VEL
LIN {X 0,Y 259.615,Z 361.811,A -85,B 0,C 180,E1 -18786.521,E2 -18786.521} C_VEL
LIN {X 0,Y 258.608,Z 399.511,A -85,B 0,C 180,E1 -18787.58,E2 -18787.58} C_VEL
LIN {X 0,Y 258.024,Z 408.887,A -85,B 0,C 180,E1 -18788.016,E2 -18788.016} C_VEL
LIN {X 0,Y 257.201,Z 418.213,A -85,B 0,C 180,E1 -18788.66,E2 -18788.66} C_VEL
LIN {X 0,Y 256.245,Z 427.438,A -85,B 0,C 180,E1 -18789.532,E2 -18789.532} C_VEL
LIN {X 0,Y 254.735,Z 438.187,A -85,B 0,C 180,E1 -18790.876,E2 -18790.876} C_VEL
LIN {X 0,Y 253.314,Z 446.445,A -85,B 0,C 180,E1 -18792.231,E2 -18792.231} C_VEL
LIN {X 0,Y 251.912,Z 454.113,A -85,B 0,C 180,E1 -18793.801,E2 -18793.801} C_VEL
LIN {X 0,Y 250.738,Z 460.423,A -85,B 0,C 180,E1 -18795.389,E2 -18795.389} C_VEL
LIN {X 0,Y 249.688,Z 465.664,A -85,B 0,C 180,E1 -18796.987,E2 -18796.987} C_VEL
LIN {X 0,Y 248.861,Z 470.033,A -85,B 0,C 180,E1 -18798.599,E2 -18798.599} C_VEL
LIN {X 0,Y 247.92,Z 475.184,A -85,B 0,C 180,E1 -18801.03,E2 -18801.03} C_VEL
LIN {X 0,Y 247.326,Z 478.964,A -85,B 0,C 180,E1 -18803.474,E2 -18803.474} C_VEL
LIN {X 0,Y 247.058,Z 480.698,A -85,B 0,C 180,E1 -18805.105,E2 -18805.105} C_VEL
LIN {X 0,Y 246.932,Z 481.939,A -85,B 0,C 180,E1 -18806.737,E2 -18806.737} C_VEL
LIN {X 0,Y 246.881,Z 482.709,A -85,B 0,C 180,E1 -18808.369,E2 -18808.369} C_VEL
LIN {X 0,Y 246.857,Z 483,A -85,B 0,C 180,E1 -18810,E2 -18810} C_VEL
LIN {X 0,Y 246.881,Z 482.702,A -85,B 0,C 180,E1 -18811.631,E2 -18811.631} C_VEL
LIN {X 0,Y 246.931,Z 481.916,A -85,B 0,C 180,E1 -18813.263,E2 -18813.263} C_VEL
LIN {X 0,Y 247.088,Z 480.132,A -85,B 0,C 180,E1 -18815.429,E2 -18815.429} C_VEL
LIN {X 0,Y 247.67,Z 476.591,A -85,B 0,C 180,E1 -18818.157,E2 -18818.157} C_VEL
LIN {X 0,Y 248.484,Z 471.855,A -85,B 0,C 180,E1 -18820.593,E2 -18820.593} C_VEL
LIN {X 0,Y 249.458,Z 466.724,A -85,B 0,C 180,E1 -18822.611,E2 -18822.611} C_VEL
LIN {X 0,Y 250.482,Z 461.706,A -85,B 0,C 180,E1 -18824.211,E2 -18824.211} C_VEL
LIN {X 0,Y 251.599,Z 455.662,A -85,B 0,C 180,E1 -18825.804,E2 -18825.804} C_VEL
LIN {X 0,Y 252.97,Z 448.304,A -85,B 0,C 180,E1 -18827.376,E2 -18827.376} C_VEL
LIN {X 0,Y 254.337,Z 440.421,A -85,B 0,C 180,E1 -18828.737,E2 -18828.737} C_VEL
LIN {X 0,Y 255.585,Z 432.085,A -85,B 0,C 180,E1 -18829.894,E2 -18829.894} C_VEL
LIN {X 0,Y 256.81,Z 421.789,A -85,B 0,C 180,E1 -18831.012,E2 -18831.012} C_VEL
LIN {X 0,Y 257.882,Z 410.092,A -85,B 0,C 180,E1 -18831.881,E2 -18831.881} C_VEL
LIN {X 0,Y 258.473,Z 401.337,A -85,B 0,C 180,E1 -18832.319,E2 -18832.319} C_VEL
LIN {X 0,Y 259.242,Z 373.503,A -85,B 0,C 180,E1 -18833.13,E2 -18833.13} C_VEL
LIN {X 0,Y 259.435,Z 359.455,A -85,B 0,C 180,E1 -18833.526,E2 -18833.526} C_VEL
LIN {X 0,Y 255.552,Z 336.884,A -85,B 0,C 180,E1 -18834.587,E2 -18834.587} C_VEL
LIN {X 0,Y 251.932,Z 326.503,A -85,B 0,C 180,E1 -18835.284,E2 -18835.284} C_VEL
LIN {X 0,Y 250.958,Z 323.684,A -85,B 0,C 180,E1 -18835.574,E2 -18835.574} C_VEL
LIN {X 0,Y 249.487,Z 316.111,A -85,B 0,C 180,E1 -18839.16,E2 -18839.16} C_VEL
LIN {X 0,Y 249.079,Z 314.359,A -85,B 0,C 180,E1 -18840.132,E2 -18840.132} C_VEL
LIN {X 0,Y 249.041,Z 314.262,A -85,B 0,C 180,E1 -18845.076,E2 -18845.076} C_VEL
LIN {X 0,Y 249.019,Z 314.278,A -85,B 0,C 180,E1 -18848.381,E2 -18848.381} C_VEL
LIN {X 0,Y 248.965,Z 314.268,A -85,B 0,C 180,E1 -18852.782,E2 -18852.782} C_VEL
LIN {X 0,Y 248.975,Z 314.277,A -85,B 0,C 180,E1 -18857.354,E2 -18857.354} C_VEL
LIN {X 0,Y 249.039,Z 314.246,A -85,B 0,C 180,E1 -18862.2,E2 -18862.2} C_VEL
LIN {X 0,Y 249.038,Z 314.274,A -85,B 0,C 180,E1 -18865.639,E2 -18865.639} C_VEL
LIN {X 0,Y 248.995,Z 314.271,A -85,B 0,C 180,E1 -18869.466,E2 -18869.466} C_VEL
LIN {X 0,Y 249.015,Z 314.279,A -85,B 0,C 180,E1 -18873.156,E2 -18873.156} C_VEL
LIN {X 0,Y 248.999,Z 314.269,A -85,B 0,C 180,E1 -18876.725,E2 -18876.725} C_VEL
LIN {X 0,Y 249.036,Z 314.272,A -85,B 0,C 180,E1 -18880.206,E2 -18880.206} C_VEL
LIN {X 0,Y 249.152,Z 314.258,A -85,B 0,C 180,E1 -18883.616,E2 -18883.616} C_VEL
LIN {X 0,Y 249.212,Z 314.25,A -85,B 0,C 180,E1 -18888.615,E2 -18888.615} C_VEL
LIN {X 0,Y 249.424,Z 314.228,A -85,B 0,C 180,E1 -18891.901,E2 -18891.901} C_VEL
LIN {X 0,Y 249.25,Z 314.23,A -85,B 0,C 180,E1 -18895.148,E2 -18895.148} C_VEL
LIN {X 0,Y 249.649,Z 314.199,A -85,B 0,C 180,E1 -18898.387,E2 -18898.387} C_VEL
LIN {X 0,Y 249.647,Z 314.2,A -85,B 0,C 180,E1 -18901.613,E2 -18901.613} C_VEL
LIN {X 0,Y 249.409,Z 314.221,A -85,B 0,C 180,E1 -18906.539,E2 -18906.539} C_VEL
LIN {X 0,Y 249.326,Z 314.241,A -85,B 0,C 180,E1 -18909.737,E2 -18909.737} C_VEL
LIN {X 0,Y 249.139,Z 314.25,A -85,B 0,C 180,E1 -18914.708,E2 -18914.708} C_VEL
LIN {X 0,Y 249.073,Z 314.271,A -85,B 0,C 180,E1 -18918.082,E2 -18918.082} C_VEL
LIN {X 0,Y 249.037,Z 314.263,A -85,B 0,C 180,E1 -18921.523,E2 -18921.523} C_VEL
LIN {X 0,Y 249.042,Z 314.276,A -85,B 0,C 180,E1 -18925.441,E2 -18925.441} C_VEL
LIN {X 0,Y 249.029,Z 314.268,A -85,B 0,C 180,E1 -18928.973,E2 -18928.973} C_VEL
LIN {X 0,Y 249.023,Z 314.276,A -85,B 0,C 180,E1 -18932.427,E2 -18932.427} C_VEL
LIN {X 0,Y 249.007,Z 314.266,A -85,B 0,C 180,E1 -18936.35,E2 -18936.35} C_VEL
LIN {X 0,Y 248.975,Z 314.254,A -85,B 0,C 180,E1 -18940.484,E2 -18940.484} C_VEL
LIN {X 0,Y 248.959,Z 314.287,A -85,B 0,C 180,E1 -18944.89,E2 -18944.89} C_VEL
LIN {X 0,Y 248.976,Z 314.266,A -85,B 0,C 180,E1 -18947.356,E2 -18947.356} C_VEL
LIN {X 0,Y 249.038,Z 314.276,A -85,B 0,C 180,E1 -18952.202,E2 -18952.202} C_VEL
LIN {X 0,Y 249.041,Z 314.262,A -85,B 0,C 180,E1 -18955.64,E2 -18955.64} C_VEL
LIN {X 0,Y 249.053,Z 314.39,A -85,B 0,C 180,E1 -18959.971,E2 -18959.971} C_VEL
LIN {X 0,Y 250.634,Z 322.088,A -85,B 0,C 180,E1 -18963.807,E2 -18963.807} C_VEL
LIN {X 0,Y 251.065,Z 324.095,A -85,B 0,C 180,E1 -18964.556,E2 -18964.556} C_VEL
LIN {X 0,Y 255.034,Z 334.962,A -85,B 0,C 180,E1 -18965.346,E2 -18965.346} C_VEL
LIN {X 0,Y 257.985,Z 350.181,A -85,B 0,C 180,E1 -18966.102,E2 -18966.102} C_VEL
LIN {X 0,Y 259.564,Z 361.233,A -85,B 0,C 180,E1 -18966.583,E2 -18966.583} C_VEL
LIN {X 0,Y 258.494,Z 399.927,A -85,B 0,C 180,E1 -18967.671,E2 -18967.671} C_VEL
LIN {X 0,Y 257.933,Z 409.04,A -85,B 0,C 180,E1 -18968.102,E2 -18968.102} C_VEL
LIN {X 0,Y 257.126,Z 419.19,A -85,B 0,C 180,E1 -18968.822,E2 -18968.822} C_VEL
LIN {X 0,Y 255.859,Z 430.257,A -85,B 0,C 180,E1 -18969.919,E2 -18969.919} C_VEL
LIN {X 0,Y 254.331,Z 440.156,A -85,B 0,C 180,E1 -18971.263,E2 -18971.263} C_VEL
LIN {X 0,Y 253.029,Z 448.083,A -85,B 0,C 180,E1 -18972.628,E2 -18972.628} C_VEL
LIN {X 0,Y 251.637,Z 455.478,A -85,B 0,C 180,E1 -18974.199,E2 -18974.199} C_VEL
LIN {X 0,Y 250.217,Z 462.969,A -85,B 0,C 180,E1 -18976.188,E2 -18976.188} C_VEL
LIN {X 0,Y 248.892,Z 469.838,A -85,B 0,C 180,E1 -18978.6,E2 -18978.6} C_VEL
LIN {X 0,Y 247.927,Z 475.032,A -85,B 0,C 180,E1 -18981.031,E2 -18981.031} C_VEL
LIN {X 0,Y 247.471,Z 477.697,A -85,B 0,C 180,E1 -18982.658,E2 -18982.658} C_VEL
LIN {X 0,Y 247.059,Z 480.616,A -85,B 0,C 180,E1 -18985.105,E2 -18985.105} C_VEL
LIN {X 0,Y 246.934,Z 481.89,A -85,B 0,C 180,E1 -18986.737,E2 -18986.737} C_VEL
LIN {X 0,Y 246.882,Z 482.693,A -85,B 0,C 180,E1 -18988.369,E2 -18988.369} C_VEL
LIN {X 0,Y 246.858,Z 482.999,A -85,B 0,C 180,E1 -18990,E2 -18990} C_VEL
LIN {X 0,Y 246.877,Z 482.718,A -85,B 0,C 180,E1 -18991.631,E2 -18991.631} C_VEL
LIN {X 0,Y 246.907,Z 481.965,A -85,B 0,C 180,E1 -18993.263,E2 -18993.263} C_VEL
LIN {X 0,Y 247.088,Z 480.217,A -85,B 0,C 180,E1 -18995.427,E2 -18995.427} C_VEL
LIN {X 0,Y 247.47,Z 477.876,A -85,B 0,C 180,E1 -18997.342,E2 -18997.342} C_VEL
LIN {X 0,Y 247.916,Z 475.267,A -85,B 0,C 180,E1 -18998.97,E2 -18998.97} C_VEL
LIN {X 0,Y 248.836,Z 470.137,A -85,B 0,C 180,E1 -19001.402,E2 -19001.402} C_VEL
LIN {X 0,Y 249.931,Z 464.619,A -85,B 0,C 180,E1 -19003.414,E2 -19003.414} C_VEL
LIN {X 0,Y 251.296,Z 457.686,A -85,B 0,C 180,E1 -19005.407,E2 -19005.407} C_VEL
LIN {X 0,Y 252.74,Z 449.727,A -85,B 0,C 180,E1 -19007.184,E2 -19007.184} C_VEL
LIN {X 0,Y 254.131,Z 442.14,A -85,B 0,C 180,E1 -19008.544,E2 -19008.544} C_VEL
LIN {X 0,Y 255.386,Z 434.186,A -85,B 0,C 180,E1 -19009.7,E2 -19009.7} C_VEL
LIN {X 0,Y 256.393,Z 425.967,A -85,B 0,C 180,E1 -19010.665,E2 -19010.665} C_VEL
LIN {X 0,Y 257.356,Z 417.56,A -85,B 0,C 180,E1 -19011.429,E2 -19011.429} C_VEL
LIN {X 0,Y 258.115,Z 407.828,A -85,B 0,C 180,E1 -19012.088,E2 -19012.088} C_VEL
LIN {X 0,Y 258.589,Z 398.203,A -85,B 0,C 180,E1 -19012.52,E2 -19012.52} C_VEL
LIN {X 0,Y 259.544,Z 359.846,A -85,B 0,C 180,E1 -19013.589,E2 -19013.589} C_VEL
LIN {X 0,Y 255.825,Z 338.009,A -85,B 0,C 180,E1 -19014.612,E2 -19014.612} C_VEL
LIN {X 0,Y 253.622,Z 330.923,A -85,B 0,C 180,E1 -19015.056,E2 -19015.056} C_VEL
LIN {X 0,Y 251.039,Z 323.975,A -85,B 0,C 180,E1 -19015.6,E2 -19015.6} C_VEL
LIN {X 0,Y 250.508,Z 321.372,A -85,B 0,C 180,E1 -19016.671,E2 -19016.671} C_VEL
LIN {X 0,Y 249.071,Z 314.357,A -85,B 0,C 180,E1 -19020.232,E2 -19020.232} C_VEL
LIN {X 0,Y 249.042,Z 314.261,A -85,B 0,C 180,E1 -19025.076,E2 -19025.076} C_VEL
LIN {X 0,Y 249.02,Z 314.278,A -85,B 0,C 180,E1 -19028.381,E2 -19028.381} C_VEL
LIN {X 0,Y 248.966,Z 314.266,A -85,B 0,C 180,E1 -19032.781,E2 -19032.781} C_VEL
LIN {X 0,Y 248.973,Z 314.279,A -85,B 0,C 180,E1 -19037.353,E2 -19037.353} C_VEL
LIN {X 0,Y 249.017,Z 314.247,A -85,B 0,C 180,E1 -19042.206,E2 -19042.206} C_VEL
LIN {X 0,Y 249.038,Z 314.274,A -85,B 0,C 180,E1 -19045.638,E2 -19045.638} C_VEL
LIN {X 0,Y 248.996,Z 314.272,A -85,B 0,C 180,E1 -19049.465,E2 -19049.465} C_VEL
LIN {X 0,Y 249.016,Z 314.279,A -85,B 0,C 180,E1 -19053.155,E2 -19053.155} C_VEL
LIN {X 0,Y 249,Z 314.27,A -85,B 0,C 180,E1 -19056.725,E2 -19056.725} C_VEL
LIN {X 0,Y 249.036,Z 314.271,A -85,B 0,C 180,E1 -19060.205,E2 -19060.205} C_VEL
LIN {X 0,Y 249.153,Z 314.258,A -85,B 0,C 180,E1 -19063.616,E2 -19063.616} C_VEL
LIN {X 0,Y 249.212,Z 314.249,A -85,B 0,C 180,E1 -19068.614,E2 -19068.614} C_VEL
LIN {X 0,Y 249.425,Z 314.228,A -85,B 0,C 180,E1 -19071.901,E2 -19071.901} C_VEL
LIN {X 0,Y 249.25,Z 314.23,A -85,B 0,C 180,E1 -19075.147,E2 -19075.147} C_VEL
LIN {X 0,Y 249.649,Z 314.199,A -85,B 0,C 180,E1 -19078.387,E2 -19078.387} C_VEL
LIN {X 0,Y 249.647,Z 314.2,A -85,B 0,C 180,E1 -19081.613,E2 -19081.613} C_VEL
LIN {X 0,Y 249.401,Z 314.223,A -85,B 0,C 180,E1 -19086.673,E2 -19086.673} C_VEL
LIN {X 0,Y 249.325,Z 314.241,A -85,B 0,C 180,E1 -19089.737,E2 -19089.737} C_VEL
LIN {X 0,Y 249.124,Z 314.249,A -85,B 0,C 180,E1 -19093.679,E2 -19093.679} C_VEL
LIN {X 0,Y 248.431,Z 314.34,A -85,B 0,C 180,E1 -19095.028,E2 -19095.028} C_VEL
LIN {X 0,Y 245.542,Z 314.71,A -85,B 0,C 180,E1 -19097.226,E2 -19097.226} C_VEL
LIN {X 0,Y 243.097,Z 315.015,A -85,B 0,C 180,E1 -19099.016,E2 -19099.016} C_VEL
LIN {X 0,Y 242.049,Z 315.139,A -85,B 0,C 180,E1 -19100.406,E2 -19100.406} C_VEL
LIN {X 0,Y 241.964,Z 315.145,A -85,B 0,C 180,E1 -19100.877,E2 -19100.877} C_VEL
LIN {X 0,Y 241.976,Z 315.151,A -85,B 0,C 180,E1 -19103.992,E2 -19103.992} C_VEL
LIN {X 0,Y 241.954,Z 315.154,A -85,B 0,C 180,E1 -19107.694,E2 -19107.694} C_VEL
LIN {X 0,Y 241.947,Z 315.156,A -85,B 0,C 180,E1 -19111.524,E2 -19111.524} C_VEL
LIN {X 0,Y 241.974,Z 315.145,A -85,B 0,C 180,E1 -19115.588,E2 -19115.588} C_VEL
LIN {X 0,Y 241.935,Z 315.122,A -85,B 0,C 180,E1 -19119.723,E2 -19119.723} C_VEL
LIN {X 0,Y 241.892,Z 315.166,A -85,B 0,C 180,E1 -19124.211,E2 -19124.211} C_VEL
LIN {X 0,Y 241.904,Z 315.138,A -85,B 0,C 180,E1 -19128.072,E2 -19128.072} C_VEL
LIN {X 0,Y 241.98,Z 315.157,A -85,B 0,C 180,E1 -19132.418,E2 -19132.418} C_VEL
LIN {X 0,Y 241.977,Z 315.15,A -85,B 0,C 180,E1 -19136.508,E2 -19136.508} C_VEL
LIN {X 0,Y 242.041,Z 315.261,A -85,B 0,C 180,E1 -19139.341,E2 -19139.341} C_VEL
LIN {X 0,Y 243.31,Z 321.276,A -85,B 0,C 180,E1 -19142.474,E2 -19142.474} C_VEL
LIN {X 0,Y 243.743,Z 323.733,A -85,B 0,C 180,E1 -19143.585,E2 -19143.585} C_VEL
LIN {X 0,Y 245.643,Z 328.709,A -85,B 0,C 180,E1 -19144.046,E2 -19144.046} C_VEL
LIN {X 0,Y 249.179,Z 338.305,A -85,B 0,C 180,E1 -19144.741,E2 -19144.741} C_VEL
LIN {X 0,Y 252.48,Z 357.144,A -85,B 0,C 180,E1 -19145.672,E2 -19145.672} C_VEL
LIN {X 0,Y 253.112,Z 362.438,A -85,B 0,C 180,E1 -19145.898,E2 -19145.898} C_VEL
LIN {X 0,Y 252.039,Z 399.992,A -85,B 0,C 180,E1 -19146.982,E2 -19146.982} C_VEL
LIN {X 0,Y 251.401,Z 409.633,A -85,B 0,C 180,E1 -19147.453,E2 -19147.453} C_VEL
LIN {X 0,Y 250.351,Z 420.599,A -85,B 0,C 180,E1 -19148.259,E2 -19148.259} C_VEL
LIN {X 0,Y 249.14,Z 430.867,A -85,B 0,C 180,E1 -19149.353,E2 -19149.353} C_VEL
LIN {X 0,Y 247.831,Z 439.421,A -85,B 0,C 180,E1 -19150.537,E2 -19150.537} C_VEL
LIN {X 0,Y 246.383,Z 447.469,A -85,B 0,C 180,E1 -19151.929,E2 -19151.929} C_VEL
LIN {X 0,Y 245.108,Z 454.116,A -85,B 0,C 180,E1 -19153.338,E2 -19153.338} C_VEL
LIN {X 0,Y 243.862,Z 460.425,A -85,B 0,C 180,E1 -19154.967,E2 -19154.967} C_VEL
LIN {X 0,Y 242.773,Z 465.665,A -85,B 0,C 180,E1 -19156.61,E2 -19156.61} C_VEL
LIN {X 0,Y 241.908,Z 470.034,A -85,B 0,C 180,E1 -19158.266,E2 -19158.266} C_VEL
LIN {X 0,Y 240.903,Z 475.185,A -85,B 0,C 180,E1 -19160.767,E2 -19160.767} C_VEL
LIN {X 0,Y 240.273,Z 478.965,A -85,B 0,C 180,E1 -19163.281,E2 -19163.281} C_VEL
LIN {X 0,Y 239.988,Z 480.699,A -85,B 0,C 180,E1 -19164.96,E2 -19164.96} C_VEL
LIN {X 0,Y 239.841,Z 481.939,A -85,B 0,C 180,E1 -19166.64,E2 -19166.64} C_VEL
LIN {X 0,Y 239.797,Z 482.709,A -85,B 0,C 180,E1 -19168.321,E2 -19168.321} C_VEL
LIN {X 0,Y 239.772,Z 483,A -85,B 0,C 180,E1 -19170,E2 -19170} C_VEL
LIN {X 0,Y 239.797,Z 482.701,A -85,B 0,C 180,E1 -19171.679,E2 -19171.679} C_VEL
LIN {X 0,Y 239.84,Z 481.916,A -85,B 0,C 180,E1 -19173.36,E2 -19173.36} C_VEL
LIN {X 0,Y 239.99,Z 480.378,A -85,B 0,C 180,E1 -19175.333,E2 -19175.333} C_VEL
LIN {X 0,Y 240.42,Z 477.759,A -85,B 0,C 180,E1 -19177.559,E2 -19177.559} C_VEL
LIN {X 0,Y 240.9,Z 475.114,A -85,B 0,C 180,E1 -19179.233,E2 -19179.233} C_VEL
LIN {X 0,Y 241.903,Z 469.941,A -85,B 0,C 180,E1 -19181.734,E2 -19181.734} C_VEL
LIN {X 0,Y 243.315,Z 463.118,A -85,B 0,C 180,E1 -19184.212,E2 -19184.212} C_VEL
LIN {X 0,Y 244.776,Z 455.659,A -85,B 0,C 180,E1 -19186.256,E2 -19186.256} C_VEL
LIN {X 0,Y 246.208,Z 448.301,A -85,B 0,C 180,E1 -19187.87,E2 -19187.87} C_VEL
LIN {X 0,Y 247.608,Z 440.417,A -85,B 0,C 180,E1 -19189.266,E2 -19189.266} C_VEL
LIN {X 0,Y 248.93,Z 432.08,A -85,B 0,C 180,E1 -19190.449,E2 -19190.449} C_VEL
LIN {X 0,Y 250.177,Z 421.952,A -85,B 0,C 180,E1 -19191.578,E2 -19191.578} C_VEL
LIN {X 0,Y 251.273,Z 410.466,A -85,B 0,C 180,E1 -19192.463,E2 -19192.463} C_VEL
LIN {X 0,Y 251.95,Z 400.829,A -85,B 0,C 180,E1 -19192.95,E2 -19192.95} C_VEL
LIN {X 0,Y 253.065,Z 362.673,A -85,B 0,C 180,E1 -19194.057,E2 -19194.057} C_VEL
LIN {X 0,Y 251.592,Z 351.567,A -85,B 0,C 180,E1 -19194.548,E2 -19194.548} C_VEL
LIN {X 0,Y 248.755,Z 337.034,A -85,B 0,C 180,E1 -19195.3,E2 -19195.3} C_VEL
LIN {X 0,Y 244.499,Z 325.989,A -85,B 0,C 180,E1 -19196.125,E2 -19196.125} C_VEL
LIN {X 0,Y 243.747,Z 323.743,A -85,B 0,C 180,E1 -19196.37,E2 -19196.37} C_VEL
LIN {X 0,Y 242.491,Z 317.271,A -85,B 0,C 180,E1 -19199.518,E2 -19199.518} C_VEL
LIN {X 0,Y 242.01,Z 315.237,A -85,B 0,C 180,E1 -19200.663,E2 -19200.663} C_VEL
LIN {X 0,Y 242.004,Z 315.139,A -85,B 0,C 180,E1 -19205.596,E2 -19205.596} C_VEL
LIN {X 0,Y 241.936,Z 315.145,A -85,B 0,C 180,E1 -19209.722,E2 -19209.722} C_VEL
LIN {X 0,Y 241.892,Z 315.162,A -85,B 0,C 180,E1 -19214.21,E2 -19214.21} C_VEL
LIN {X 0,Y 241.903,Z 315.152,A -85,B 0,C 180,E1 -19218.071,E2 -19218.071} C_VEL
LIN {X 0,Y 241.978,Z 315.125,A -85,B 0,C 180,E1 -19222.416,E2 -19222.416} C_VEL
LIN {X 0,Y 241.974,Z 315.156,A -85,B 0,C 180,E1 -19226.507,E2 -19226.507} C_VEL
LIN {X 0,Y 241.97,Z 315.144,A -85,B 0,C 180,E1 -19230.613,E2 -19230.613} C_VEL
LIN {X 0,Y 241.991,Z 315.154,A -85,B 0,C 180,E1 -19234.197,E2 -19234.197} C_VEL
LIN {X 0,Y 241.979,Z 315.14,A -85,B 0,C 180,E1 -19238.338,E2 -19238.338} C_VEL
LIN {X 0,Y 242.1,Z 315.136,A -85,B 0,C 180,E1 -19243.324,E2 -19243.324} C_VEL
LIN {X 0,Y 242.145,Z 315.126,A -85,B 0,C 180,E1 -19248.278,E2 -19248.278} C_VEL
LIN {X 0,Y 242.374,Z 315.105,A -85,B 0,C 180,E1 -19251.664,E2 -19251.664} C_VEL
LIN {X 0,Y 242.393,Z 315.096,A -85,B 0,C 180,E1 -19253.34,E2 -19253.34} C_VEL
LIN {X 0,Y 242.609,Z 315.075,A -85,B 0,C 180,E1 -19258.34,E2 -19258.34} C_VEL
LIN {X 0,Y 242.607,Z 315.076,A -85,B 0,C 180,E1 -19261.66,E2 -19261.66} C_VEL
LIN {X 0,Y 242.384,Z 315.097,A -85,B 0,C 180,E1 -19266.66,E2 -19266.66} C_VEL
LIN {X 0,Y 242.254,Z 315.12,A -85,B 0,C 180,E1 -19270.024,E2 -19270.024} C_VEL
LIN {X 0,Y 242.098,Z 315.128,A -85,B 0,C 180,E1 -19275.145,E2 -19275.145} C_VEL
LIN {X 0,Y 242.011,Z 315.15,A -85,B 0,C 180,E1 -19278.629,E2 -19278.629} C_VEL
LIN {X 0,Y 241.967,Z 315.14,A -85,B 0,C 180,E1 -19282.185,E2 -19282.185} C_VEL
LIN {X 0,Y 241.982,Z 315.155,A -85,B 0,C 180,E1 -19285.827,E2 -19285.827} C_VEL
LIN {X 0,Y 241.963,Z 315.145,A -85,B 0,C 180,E1 -19289.589,E2 -19289.589} C_VEL
LIN {X 0,Y 241.975,Z 315.156,A -85,B 0,C 180,E1 -19293.494,E2 -19293.494} C_VEL
LIN {X 0,Y 241.979,Z 315.125,A -85,B 0,C 180,E1 -19297.584,E2 -19297.584} C_VEL
LIN {X 0,Y 241.904,Z 315.151,A -85,B 0,C 180,E1 -19301.93,E2 -19301.93} C_VEL
LIN {X 0,Y 241.897,Z 315.153,A -85,B 0,C 180,E1 -19306.581,E2 -19306.581} C_VEL
LIN {X 0,Y 241.99,Z 315.153,A -85,B 0,C 180,E1 -19311.642,E2 -19311.642} C_VEL
LIN {X 0,Y 241.984,Z 315.142,A -85,B 0,C 180,E1 -19314.49,E2 -19314.49} C_VEL
LIN {X 0,Y 241.993,Z 315.189,A -85,B 0,C 180,E1 -19319.213,E2 -19319.213} C_VEL
LIN {X 0,Y 242.002,Z 315.294,A -85,B 0,C 180,E1 -19319.456,E2 -19319.456} C_VEL
LIN {X 0,Y 243.644,Z 323.279,A -85,B 0,C 180,E1 -19323.515,E2 -19323.515} C_VEL
LIN {X 0,Y 243.851,Z 324.071,A -85,B 0,C 180,E1 -19323.743,E2 -19323.743} C_VEL
LIN {X 0,Y 248.692,Z 336.834,A -85,B 0,C 180,E1 -19324.732,E2 -19324.732} C_VEL
LIN {X 0,Y 251.138,Z 348.929,A -85,B 0,C 180,E1 -19325.369,E2 -19325.369} C_VEL
LIN {X 0,Y 253.07,Z 361.68,A -85,B 0,C 180,E1 -19325.958,E2 -19325.958} C_VEL
LIN {X 0,Y 251.925,Z 400.494,A -85,B 0,C 180,E1 -19327.079,E2 -19327.079} C_VEL
LIN {X 0,Y 251.284,Z 410.3,A -85,B 0,C 180,E1 -19327.572,E2 -19327.572} C_VEL
LIN {X 0,Y 250.286,Z 421.411,A -85,B 0,C 180,E1 -19328.419,E2 -19328.419} C_VEL
LIN {X 0,Y 249,Z 431.767,A -85,B 0,C 180,E1 -19329.557,E2 -19329.557} C_VEL
LIN {X 0,Y 247.635,Z 440.16,A -85,B 0,C 180,E1 -19330.736,E2 -19330.736} C_VEL
LIN {X 0,Y 246.263,Z 448.087,A -85,B 0,C 180,E1 -19332.135,E2 -19332.135} C_VEL
LIN {X 0,Y 245.138,Z 453.779,A -85,B 0,C 180,E1 -19333.34,E2 -19333.34} C_VEL
LIN {X 0,Y 243.888,Z 460.138,A -85,B 0,C 180,E1 -19334.969,E2 -19334.969} C_VEL
LIN {X 0,Y 242.791,Z 465.425,A -85,B 0,C 180,E1 -19336.611,E2 -19336.611} C_VEL
LIN {X 0,Y 241.943,Z 469.84,A -85,B 0,C 180,E1 -19338.268,E2 -19338.268} C_VEL
LIN {X 0,Y 240.91,Z 475.033,A -85,B 0,C 180,E1 -19340.767,E2 -19340.767} C_VEL
LIN {X 0,Y 240.422,Z 477.698,A -85,B 0,C 180,E1 -19342.441,E2 -19342.441} C_VEL
LIN {X 0,Y 239.969,Z 480.617,A -85,B 0,C 180,E1 -19344.96,E2 -19344.96} C_VEL
LIN {X 0,Y 239.843,Z 481.89,A -85,B 0,C 180,E1 -19346.64,E2 -19346.64} C_VEL
LIN {X 0,Y 239.798,Z 482.693,A -85,B 0,C 180,E1 -19348.321,E2 -19348.321} C_VEL
LIN {X 0,Y 239.772,Z 482.999,A -85,B 0,C 180,E1 -19350,E2 -19350} C_VEL
LIN {X 0,Y 239.792,Z 482.718,A -85,B 0,C 180,E1 -19351.679,E2 -19351.679} C_VEL
LIN {X 0,Y 239.818,Z 481.965,A -85,B 0,C 180,E1 -19353.36,E2 -19353.36} C_VEL
LIN {X 0,Y 239.985,Z 480.478,A -85,B 0,C 180,E1 -19355.315,E2 -19355.315} C_VEL
LIN {X 0,Y 240.421,Z 477.875,A -85,B 0,C 180,E1 -19357.559,E2 -19357.559} C_VEL
LIN {X 0,Y 240.897,Z 475.266,A -85,B 0,C 180,E1 -19359.233,E2 -19359.233} C_VEL
LIN {X 0,Y 241.882,Z 470.135,A -85,B 0,C 180,E1 -19361.735,E2 -19361.735} C_VEL
LIN {X 0,Y 243.022,Z 464.617,A -85,B 0,C 180,E1 -19363.803,E2 -19363.803} C_VEL
LIN {X 0,Y 244.43,Z 457.683,A -85,B 0,C 180,E1 -19365.851,E2 -19365.851} C_VEL
LIN {X 0,Y 245.985,Z 449.724,A -85,B 0,C 180,E1 -19367.671,E2 -19367.671} C_VEL
LIN {X 0,Y 247.408,Z 442.135,A -85,B 0,C 180,E1 -19369.067,E2 -19369.067} C_VEL
LIN {X 0,Y 248.724,Z 434.181,A -85,B 0,C 180,E1 -19370.251,E2 -19370.251} C_VEL
LIN {X 0,Y 249.78,Z 425.961,A -85,B 0,C 180,E1 -19371.239,E2 -19371.239} C_VEL
LIN {X 0,Y 250.678,Z 418.528,A -85,B 0,C 180,E1 -19371.942,E2 -19371.942} C_VEL
LIN {X 0,Y 251.418,Z 408.999,A -85,B 0,C 180,E1 -19372.631,E2 -19372.631} C_VEL
LIN {X 0,Y 251.979,Z 399.767,A -85,B 0,C 180,E1 -19373.078,E2 -19373.078} C_VEL
LIN {X 0,Y 253.048,Z 360.849,A -85,B 0,C 180,E1 -19374.202,E2 -19374.202} C_VEL
LIN {X 0,Y 249.543,Z 340.06,A -85,B 0,C 180,E1 -19375.21,E2 -19375.21} C_VEL
LIN {X 0,Y 247.597,Z 333.705,A -85,B 0,C 180,E1 -19375.622,E2 -19375.622} C_VEL
LIN {X 0,Y 243.777,Z 323.893,A -85,B 0,C 180,E1 -19376.428,E2 -19376.428} C_VEL
LIN {X 0,Y 242.927,Z 319.418,A -85,B 0,C 180,E1 -19378.512,E2 -19378.512} C_VEL
LIN {X 0,Y 242.047,Z 315.225,A -85,B 0,C 180,E1 -19380.779,E2 -19380.779} C_VEL
LIN {X 0,Y 241.976,Z 315.142,A -85,B 0,C 180,E1 -19385.586,E2 -19385.586} C_VEL
LIN {X 0,Y 241.937,Z 315.147,A -85,B 0,C 180,E1 -19389.722,E2 -19389.722} C_VEL
LIN {X 0,Y 241.893,Z 315.162,A -85,B 0,C 180,E1 -19394.209,E2 -19394.209} C_VEL
LIN {X 0,Y 241.901,Z 315.154,A -85,B 0,C 180,E1 -19398.07,E2 -19398.07} C_VEL
LIN {X 0,Y 241.96,Z 315.125,A -85,B 0,C 180,E1 -19402.413,E2 -19402.413} C_VEL
LIN {X 0,Y 241.975,Z 315.156,A -85,B 0,C 180,E1 -19406.506,E2 -19406.506} C_VEL
LIN {X 0,Y 241.971,Z 315.144,A -85,B 0,C 180,E1 -19410.613,E2 -19410.613} C_VEL
LIN {X 0,Y 241.992,Z 315.154,A -85,B 0,C 180,E1 -19414.196,E2 -19414.196} C_VEL
LIN {X 0,Y 241.98,Z 315.14,A -85,B 0,C 180,E1 -19418.338,E2 -19418.338} C_VEL
LIN {X 0,Y 242.101,Z 315.137,A -85,B 0,C 180,E1 -19423.324,E2 -19423.324} C_VEL
LIN {X 0,Y 242.146,Z 315.125,A -85,B 0,C 180,E1 -19428.278,E2 -19428.278} C_VEL
LIN {X 0,Y 242.375,Z 315.105,A -85,B 0,C 180,E1 -19431.664,E2 -19431.664} C_VEL
LIN {X 0,Y 242.393,Z 315.096,A -85,B 0,C 180,E1 -19433.34,E2 -19433.34} C_VEL
LIN {X 0,Y 242.609,Z 315.075,A -85,B 0,C 180,E1 -19438.34,E2 -19438.34} C_VEL
LIN {X 0,Y 242.607,Z 315.076,A -85,B 0,C 180,E1 -19441.66,E2 -19441.66} C_VEL
LIN {X 0,Y 242.384,Z 315.097,A -85,B 0,C 180,E1 -19446.66,E2 -19446.66} C_VEL
LIN {X 0,Y 242.253,Z 315.12,A -85,B 0,C 180,E1 -19450.024,E2 -19450.024} C_VEL
LIN {X 0,Y 242.097,Z 315.128,A -85,B 0,C 180,E1 -19455.145,E2 -19455.145} C_VEL
LIN {X 0,Y 242.011,Z 315.15,A -85,B 0,C 180,E1 -19458.629,E2 -19458.629} C_VEL
LIN {X 0,Y 241.964,Z 315.145,A -85,B 0,C 180,E1 -19460.877,E2 -19460.877} C_VEL
LIN {X 0,Y 241.283,Z 315.228,A -85,B 0,C 180,E1 -19462.266,E2 -19462.266} C_VEL
LIN {X 0,Y 238.394,Z 315.598,A -85,B 0,C 180,E1 -19464.531,E2 -19464.531} C_VEL
LIN {X 0,Y 235.961,Z 315.904,A -85,B 0,C 180,E1 -19466.377,E2 -19466.377} C_VEL
LIN {X 0,Y 234.946,Z 316.026,A -85,B 0,C 180,E1 -19467.811,E2 -19467.811} C_VEL
LIN {X 0,Y 234.879,Z 316.03,A -85,B 0,C 180,E1 -19468.297,E2 -19468.297} C_VEL
LIN {X 0,Y 234.948,Z 316.03,A -85,B 0,C 180,E1 -19472.577,E2 -19472.577} C_VEL
LIN {X 0,Y 234.91,Z 316.01,A -85,B 0,C 180,E1 -19476.752,E2 -19476.752} C_VEL
LIN {X 0,Y 234.908,Z 315.992,A -85,B 0,C 180,E1 -19478.936,E2 -19478.936} C_VEL
LIN {X 0,Y 234.849,Z 316.044,A -85,B 0,C 180,E1 -19483.495,E2 -19483.495} C_VEL
LIN {X 0,Y 234.849,Z 316.029,A -85,B 0,C 180,E1 -19486.506,E2 -19486.506} C_VEL
LIN {X 0,Y 234.915,Z 316.029,A -85,B 0,C 180,E1 -19491.079,E2 -19491.079} C_VEL
LIN {X 0,Y 234.922,Z 316.018,A -85,B 0,C 180,E1 -19495.362,E2 -19495.362} C_VEL
LIN {X 0,Y 235.007,Z 316.207,A -85,B 0,C 180,E1 -19498.82,E2 -19498.82} C_VEL
LIN {X 0,Y 236.557,Z 323.653,A -85,B 0,C 180,E1 -19502.699,E2 -19502.699} C_VEL
LIN {X 0,Y 238.044,Z 327.576,A -85,B 0,C 180,E1 -19503.114,E2 -19503.114} C_VEL
LIN {X 0,Y 242.933,Z 340.377,A -85,B 0,C 180,E1 -19504.11,E2 -19504.11} C_VEL
LIN {X 0,Y 246.041,Z 358.159,A -85,B 0,C 180,E1 -19505.024,E2 -19505.024} C_VEL
LIN {X 0,Y 246.62,Z 363.792,A -85,B 0,C 180,E1 -19505.263,E2 -19505.263} C_VEL
LIN {X 0,Y 245.54,Z 400.022,A -85,B 0,C 180,E1 -19506.337,E2 -19506.337} C_VEL
LIN {X 0,Y 244.852,Z 409.769,A -85,B 0,C 180,E1 -19506.824,E2 -19506.824} C_VEL
LIN {X 0,Y 243.756,Z 420.896,A -85,B 0,C 180,E1 -19507.668,E2 -19507.668} C_VEL
LIN {X 0,Y 242.521,Z 430.872,A -85,B 0,C 180,E1 -19508.763,E2 -19508.763} C_VEL
LIN {X 0,Y 241.166,Z 439.424,A -85,B 0,C 180,E1 -19509.976,E2 -19509.976} C_VEL
LIN {X 0,Y 239.655,Z 447.472,A -85,B 0,C 180,E1 -19511.403,E2 -19511.403} C_VEL
LIN {X 0,Y 238.321,Z 454.118,A -85,B 0,C 180,E1 -19512.849,E2 -19512.849} C_VEL
LIN {X 0,Y 237.001,Z 460.427,A -85,B 0,C 180,E1 -19514.521,E2 -19514.521} C_VEL
LIN {X 0,Y 235.871,Z 465.667,A -85,B 0,C 180,E1 -19516.21,E2 -19516.21} C_VEL
LIN {X 0,Y 234.943,Z 470.036,A -85,B 0,C 180,E1 -19517.913,E2 -19517.913} C_VEL
LIN {X 0,Y 233.876,Z 475.187,A -85,B 0,C 180,E1 -19520.487,E2 -19520.487} C_VEL
LIN {X 0,Y 233.217,Z 478.966,A -85,B 0,C 180,E1 -19523.077,E2 -19523.077} C_VEL
LIN {X 0,Y 232.919,Z 480.699,A -85,B 0,C 180,E1 -19524.807,E2 -19524.807} C_VEL
LIN {X 0,Y 232.754,Z 481.94,A -85,B 0,C 180,E1 -19526.538,E2 -19526.538} C_VEL
LIN {X 0,Y 232.696,Z 482.709,A -85,B 0,C 180,E1 -19528.269,E2 -19528.269} C_VEL
LIN {X 0,Y 232.688,Z 483,A -85,B 0,C 180,E1 -19530,E2 -19530} C_VEL
LIN {X 0,Y 232.696,Z 482.701,A -85,B 0,C 180,E1 -19531.731,E2 -19531.731} C_VEL
LIN {X 0,Y 232.752,Z 481.916,A -85,B 0,C 180,E1 -19533.462,E2 -19533.462} C_VEL
LIN {X 0,Y 232.88,Z 480.659,A -85,B 0,C 180,E1 -19535.194,E2 -19535.194} C_VEL
LIN {X 0,Y 233.372,Z 477.758,A -85,B 0,C 180,E1 -19537.788,E2 -19537.788} C_VEL
LIN {X 0,Y 233.872,Z 475.112,A -85,B 0,C 180,E1 -19539.513,E2 -19539.513} C_VEL
LIN {X 0,Y 234.939,Z 469.939,A -85,B 0,C 180,E1 -19542.087,E2 -19542.087} C_VEL
LIN {X 0,Y 236.446,Z 463.116,A -85,B 0,C 180,E1 -19544.634,E2 -19544.634} C_VEL
LIN {X 0,Y 237.976,Z 455.657,A -85,B 0,C 180,E1 -19546.734,E2 -19546.734} C_VEL
LIN {X 0,Y 239.467,Z 448.298,A -85,B 0,C 180,E1 -19548.39,E2 -19548.39} C_VEL
LIN {X 0,Y 240.929,Z 440.413,A -85,B 0,C 180,E1 -19549.822,E2 -19549.822} C_VEL
LIN {X 0,Y 242.291,Z 432.076,A -85,B 0,C 180,E1 -19551.035,E2 -19551.035} C_VEL
LIN {X 0,Y 243.563,Z 422.092,A -85,B 0,C 180,E1 -19552.178,E2 -19552.178} C_VEL
LIN {X 0,Y 244.698,Z 410.783,A -85,B 0,C 180,E1 -19553.079,E2 -19553.079} C_VEL
LIN {X 0,Y 245.428,Z 400.975,A -85,B 0,C 180,E1 -19553.589,E2 -19553.589} C_VEL
LIN {X 0,Y 246.386,Z 368.947,A -85,B 0,C 180,E1 -19554.555,E2 -19554.555} C_VEL
LIN {X 0,Y 246.504,Z 361.374,A -85,B 0,C 180,E1 -19554.78,E2 -19554.78} C_VEL
LIN {X 0,Y 242.864,Z 340.293,A -85,B 0,C 180,E1 -19555.853,E2 -19555.853} C_VEL
LIN {X 0,Y 238.743,Z 329.329,A -85,B 0,C 180,E1 -19556.694,E2 -19556.694} C_VEL
LIN {X 0,Y 236.596,Z 323.792,A -85,B 0,C 180,E1 -19557.217,E2 -19557.217} C_VEL
LIN {X 0,Y 235.201,Z 317.269,A -85,B 0,C 180,E1 -19560.528,E2 -19560.528} C_VEL
LIN {X 0,Y 234.949,Z 316.093,A -85,B 0,C 180,E1 -19561.314,E2 -19561.314} C_VEL
LIN {X 0,Y 234.936,Z 316.023,A -85,B 0,C 180,E1 -19566.129,E2 -19566.129} C_VEL
LIN {X 0,Y 234.909,Z 316.028,A -85,B 0,C 180,E1 -19568.935,E2 -19568.935} C_VEL
LIN {X 0,Y 234.849,Z 316.03,A -85,B 0,C 180,E1 -19573.494,E2 -19573.494} C_VEL
LIN {X 0,Y 234.849,Z 316.044,A -85,B 0,C 180,E1 -19576.505,E2 -19576.505} C_VEL
LIN {X 0,Y 234.914,Z 315.992,A -85,B 0,C 180,E1 -19581.078,E2 -19581.078} C_VEL
LIN {X 0,Y 234.918,Z 316.033,A -85,B 0,C 180,E1 -19585.36,E2 -19585.36} C_VEL
LIN {X 0,Y 234.893,Z 316.027,A -85,B 0,C 180,E1 -19589.427,E2 -19589.427} C_VEL
LIN {X 0,Y 234.936,Z 316.032,A -85,B 0,C 180,E1 -19593.82,E2 -19593.82} C_VEL
LIN {X 0,Y 234.929,Z 316.022,A -85,B 0,C 180,E1 -19598.962,E2 -19598.962} C_VEL
LIN {X 0,Y 235.044,Z 316.016,A -85,B 0,C 180,E1 -19603.098,E2 -19603.098} C_VEL
LIN {X 0,Y 235.077,Z 316.003,A -85,B 0,C 180,E1 -19607.92,E2 -19607.92} C_VEL
LIN {X 0,Y 235.309,Z 315.984,A -85,B 0,C 180,E1 -19611.412,E2 -19611.412} C_VEL
LIN {X 0,Y 235.345,Z 315.974,A -85,B 0,C 180,E1 -19613.14,E2 -19613.14} C_VEL
LIN {X 0,Y 235.568,Z 315.951,A -85,B 0,C 180,E1 -19618.291,E2 -19618.291} C_VEL
LIN {X 0,Y 235.566,Z 315.952,A -85,B 0,C 180,E1 -19621.71,E2 -19621.71} C_VEL
LIN {X 0,Y 235.335,Z 315.975,A -85,B 0,C 180,E1 -19626.861,E2 -19626.861} C_VEL
LIN {X 0,Y 235.178,Z 315.999,A -85,B 0,C 180,E1 -19630.329,E2 -19630.329} C_VEL
LIN {X 0,Y 235.035,Z 316.01,A -85,B 0,C 180,E1 -19635.612,E2 -19635.612} C_VEL
LIN {X 0,Y 234.953,Z 316.031,A -85,B 0,C 180,E1 -19639.21,E2 -19639.21} C_VEL
LIN {X 0,Y 234.911,Z 316.02,A -85,B 0,C 180,E1 -19642.888,E2 -19642.888} C_VEL
LIN {X 0,Y 234.92,Z 316.034,A -85,B 0,C 180,E1 -19646.664,E2 -19646.664} C_VEL
LIN {X 0,Y 234.894,Z 316.027,A -85,B 0,C 180,E1 -19650.573,E2 -19650.573} C_VEL
LIN {X 0,Y 234.918,Z 316.033,A -85,B 0,C 180,E1 -19654.64,E2 -19654.64} C_VEL
LIN {X 0,Y 234.909,Z 315.993,A -85,B 0,C 180,E1 -19658.936,E2 -19658.936} C_VEL
LIN {X 0,Y 234.85,Z 316.044,A -85,B 0,C 180,E1 -19663.495,E2 -19663.495} C_VEL
LIN {X 0,Y 234.85,Z 316.031,A -85,B 0,C 180,E1 -19666.507,E2 -19666.507} C_VEL
LIN {X 0,Y 234.916,Z 316.027,A -85,B 0,C 180,E1 -19671.079,E2 -19671.079} C_VEL
LIN {X 0,Y 234.927,Z 316.017,A -85,B 0,C 180,E1 -19675.362,E2 -19675.362} C_VEL
LIN {X 0,Y 234.954,Z 316.236,A -85,B 0,C 180,E1 -19678.937,E2 -19678.937} C_VEL
LIN {X 0,Y 236.482,Z 323.582,A -85,B 0,C 180,E1 -19682.752,E2 -19682.752} C_VEL
LIN {X 0,Y 237.091,Z 325.553,A -85,B 0,C 180,E1 -19683.022,E2 -19683.022} C_VEL
LIN {X 0,Y 242.271,Z 338.406,A -85,B 0,C 180,E1 -19684.063,E2 -19684.063} C_VEL
LIN {X 0,Y 244.076,Z 346.35,A -85,B 0,C 180,E1 -19684.523,E2 -19684.523} C_VEL
LIN {X 0,Y 246.572,Z 362.205,A -85,B 0,C 180,E1 -19685.298,E2 -19685.298} C_VEL
LIN {X 0,Y 245.429,Z 399.937,A -85,B 0,C 180,E1 -19686.411,E2 -19686.411} C_VEL
LIN {X 0,Y 244.789,Z 409.687,A -85,B 0,C 180,E1 -19686.902,E2 -19686.902} C_VEL
LIN {X 0,Y 243.864,Z 420.094,A -85,B 0,C 180,E1 -19687.691,E2 -19687.691} C_VEL
LIN {X 0,Y 242.578,Z 430.268,A -85,B 0,C 180,E1 -19688.768,E2 -19688.768} C_VEL
LIN {X 0,Y 240.965,Z 440.164,A -85,B 0,C 180,E1 -19690.181,E2 -19690.181} C_VEL
LIN {X 0,Y 239.52,Z 448.09,A -85,B 0,C 180,E1 -19691.614,E2 -19691.614} C_VEL
LIN {X 0,Y 238.354,Z 453.782,A -85,B 0,C 180,E1 -19692.852,E2 -19692.852} C_VEL
LIN {X 0,Y 237.03,Z 460.141,A -85,B 0,C 180,E1 -19694.523,E2 -19694.523} C_VEL
LIN {X 0,Y 235.886,Z 465.427,A -85,B 0,C 180,E1 -19696.211,E2 -19696.211} C_VEL
LIN {X 0,Y 235,Z 469.841,A -85,B 0,C 180,E1 -19697.916,E2 -19697.916} C_VEL
LIN {X 0,Y 233.887,Z 475.034,A -85,B 0,C 180,E1 -19700.487,E2 -19700.487} C_VEL
LIN {X 0,Y 233.374,Z 477.699,A -85,B 0,C 180,E1 -19702.212,E2 -19702.212} C_VEL
LIN {X 0,Y 232.881,Z 480.617,A -85,B 0,C 180,E1 -19704.806,E2 -19704.806} C_VEL
LIN {X 0,Y 232.755,Z 481.891,A -85,B 0,C 180,E1 -19706.538,E2 -19706.538} C_VEL
LIN {X 0,Y 232.698,Z 482.693,A -85,B 0,C 180,E1 -19708.269,E2 -19708.269} C_VEL
LIN {X 0,Y 232.689,Z 482.999,A -85,B 0,C 180,E1 -19710,E2 -19710} C_VEL
LIN {X 0,Y 232.691,Z 482.718,A -85,B 0,C 180,E1 -19711.731,E2 -19711.731} C_VEL
LIN {X 0,Y 232.732,Z 481.965,A -85,B 0,C 180,E1 -19713.462,E2 -19713.462} C_VEL
LIN {X 0,Y 232.881,Z 480.741,A -85,B 0,C 180,E1 -19715.194,E2 -19715.194} C_VEL
LIN {X 0,Y 233.373,Z 477.874,A -85,B 0,C 180,E1 -19717.788,E2 -19717.788} C_VEL
LIN {X 0,Y 233.867,Z 475.265,A -85,B 0,C 180,E1 -19719.513,E2 -19719.513} C_VEL
LIN {X 0,Y 234.904,Z 470.134,A -85,B 0,C 180,E1 -19722.089,E2 -19722.089} C_VEL
LIN {X 0,Y 236.134,Z 464.615,A -85,B 0,C 180,E1 -19724.214,E2 -19724.214} C_VEL
LIN {X 0,Y 237.599,Z 457.681,A -85,B 0,C 180,E1 -19726.32,E2 -19726.32} C_VEL
LIN {X 0,Y 239.235,Z 449.72,A -85,B 0,C 180,E1 -19728.187,E2 -19728.187} C_VEL
LIN {X 0,Y 240.704,Z 442.131,A -85,B 0,C 180,E1 -19729.619,E2 -19729.619} C_VEL
LIN {X 0,Y 242.089,Z 434.176,A -85,B 0,C 180,E1 -19730.831,E2 -19730.831} C_VEL
LIN {X 0,Y 243.194,Z 425.955,A -85,B 0,C 180,E1 -19731.843,E2 -19731.843} C_VEL
LIN {X 0,Y 244.237,Z 417.126,A -85,B 0,C 180,E1 -19732.68,E2 -19732.68} C_VEL
LIN {X 0,Y 245,Z 407.732,A -85,B 0,C 180,E1 -19733.343,E2 -19733.343} C_VEL
LIN {X 0,Y 245.555,Z 398.002,A -85,B 0,C 180,E1 -19733.794,E2 -19733.794} C_VEL
LIN {X 0,Y 246.604,Z 361.831,A -85,B 0,C 180,E1 -19734.845,E2 -19734.845} C_VEL
LIN {X 0,Y 243.14,Z 341.203,A -85,B 0,C 180,E1 -19735.884,E2 -19735.884} C_VEL
LIN {X 0,Y 239.22,Z 330.36,A -85,B 0,C 180,E1 -19736.697,E2 -19736.697} C_VEL
LIN {X 0,Y 236.631,Z 323.931,A -85,B 0,C 180,E1 -19737.286,E2 -19737.286} C_VEL
LIN {X 0,Y 236.096,Z 321.368,A -85,B 0,C 180,E1 -19738.442,E2 -19738.442} C_VEL
LIN {X 0,Y 234.987,Z 316.119,A -85,B 0,C 180,E1 -19741.308,E2 -19741.308} C_VEL
LIN {X 0,Y 234.919,Z 316.024,A -85,B 0,C 180,E1 -19746.123,E2 -19746.123} C_VEL
LIN {X 0,Y 234.91,Z 316.03,A -85,B 0,C 180,E1 -19748.934,E2 -19748.934} C_VEL
LIN {X 0,Y 234.85,Z 316.028,A -85,B 0,C 180,E1 -19753.493,E2 -19753.493} C_VEL
LIN {X 0,Y 234.849,Z 316.044,A -85,B 0,C 180,E1 -19756.505,E2 -19756.505} C_VEL
LIN {X 0,Y 234.915,Z 315.992,A -85,B 0,C 180,E1 -19761.078,E2 -19761.078} C_VEL
LIN {X 0,Y 234.918,Z 316.031,A -85,B 0,C 180,E1 -19765.36,E2 -19765.36} C_VEL
LIN {X 0,Y 234.894,Z 316.028,A -85,B 0,C 180,E1 -19769.427,E2 -19769.427} C_VEL
LIN {X 0,Y 234.936,Z 316.032,A -85,B 0,C 180,E1 -19773.82,E2 -19773.82} C_VEL
LIN {X 0,Y 234.93,Z 316.021,A -85,B 0,C 180,E1 -19778.962,E2 -19778.962} C_VEL
LIN {X 0,Y 235.044,Z 316.016,A -85,B 0,C 180,E1 -19783.097,E2 -19783.097} C_VEL
LIN {X 0,Y 235.078,Z 316.003,A -85,B 0,C 180,E1 -19787.92,E2 -19787.92} C_VEL
LIN {X 0,Y 235.309,Z 315.984,A -85,B 0,C 180,E1 -19791.411,E2 -19791.411} C_VEL
LIN {X 0,Y 235.345,Z 315.974,A -85,B 0,C 180,E1 -19793.139,E2 -19793.139} C_VEL
LIN {X 0,Y 235.568,Z 315.951,A -85,B 0,C 180,E1 -19798.29,E2 -19798.29} C_VEL
LIN {X 0,Y 235.566,Z 315.952,A -85,B 0,C 180,E1 -19801.709,E2 -19801.709} C_VEL
LIN {X 0,Y 235.334,Z 315.975,A -85,B 0,C 180,E1 -19806.86,E2 -19806.86} C_VEL
LIN {X 0,Y 235.178,Z 315.999,A -85,B 0,C 180,E1 -19810.329,E2 -19810.329} C_VEL
LIN {X 0,Y 235.035,Z 316.01,A -85,B 0,C 180,E1 -19815.612,E2 -19815.612} C_VEL
LIN {X 0,Y 234.952,Z 316.031,A -85,B 0,C 180,E1 -19819.21,E2 -19819.21} C_VEL
LIN {X 0,Y 234.911,Z 316.021,A -85,B 0,C 180,E1 -19822.888,E2 -19822.888} C_VEL
LIN {X 0,Y 234.92,Z 316.034,A -85,B 0,C 180,E1 -19826.663,E2 -19826.663} C_VEL
LIN {X 0,Y 234.879,Z 316.03,A -85,B 0,C 180,E1 -19828.297,E2 -19828.297} C_VEL
LIN {X 0,Y 234.252,Z 316.114,A -85,B 0,C 180,E1 -19829.728,E2 -19829.728} C_VEL
LIN {X 0,Y 231.42,Z 316.48,A -85,B 0,C 180,E1 -19832.062,E2 -19832.062} C_VEL
LIN {X 0,Y 228.989,Z 316.781,A -85,B 0,C 180,E1 -19833.966,E2 -19833.966} C_VEL
LIN {X 0,Y 227.944,Z 316.896,A -85,B 0,C 180,E1 -19835.443,E2 -19835.443} C_VEL
LIN {X 0,Y 227.86,Z 316.899,A -85,B 0,C 180,E1 -19835.944,E2 -19835.944} C_VEL
LIN {X 0,Y 227.796,Z 316.884,A -85,B 0,C 180,E1 -19840.383,E2 -19840.383} C_VEL
LIN {X 0,Y 227.806,Z 316.918,A -85,B 0,C 180,E1 -19845.2,E2 -19845.2} C_VEL
LIN {X 0,Y 227.796,Z 316.895,A -85,B 0,C 180,E1 -19849.618,E2 -19849.618} C_VEL
LIN {X 0,Y 227.862,Z 316.9,A -85,B 0,C 180,E1 -19854.126,E2 -19854.126} C_VEL
LIN {X 0,Y 227.948,Z 317.068,A -85,B 0,C 180,E1 -19858.196,E2 -19858.196} C_VEL
LIN {X 0,Y 229.368,Z 323.67,A -85,B 0,C 180,E1 -19861.773,E2 -19861.773} C_VEL
LIN {X 0,Y 231.051,Z 328.038,A -85,B 0,C 180,E1 -19862.246,E2 -19862.246} C_VEL
LIN {X 0,Y 236.561,Z 341.868,A -85,B 0,C 180,E1 -19863.408,E2 -19863.408} C_VEL
LIN {X 0,Y 239.64,Z 359.095,A -85,B 0,C 180,E1 -19864.338,E2 -19864.338} C_VEL
LIN {X 0,Y 240.161,Z 365.031,A -85,B 0,C 180,E1 -19864.591,E2 -19864.591} C_VEL
LIN {X 0,Y 239.064,Z 400.137,A -85,B 0,C 180,E1 -19865.659,E2 -19865.659} C_VEL
LIN {X 0,Y 238.332,Z 409.938,A -85,B 0,C 180,E1 -19866.162,E2 -19866.162} C_VEL
LIN {X 0,Y 237.172,Z 421.343,A -85,B 0,C 180,E1 -19867.06,E2 -19867.06} C_VEL
LIN {X 0,Y 235.929,Z 430.876,A -85,B 0,C 180,E1 -19868.139,E2 -19868.139} C_VEL
LIN {X 0,Y 234.512,Z 439.428,A -85,B 0,C 180,E1 -19869.383,E2 -19869.383} C_VEL
LIN {X 0,Y 232.923,Z 447.475,A -85,B 0,C 180,E1 -19870.845,E2 -19870.845} C_VEL
LIN {X 0,Y 231.547,Z 454.121,A -85,B 0,C 180,E1 -19872.331,E2 -19872.331} C_VEL
LIN {X 0,Y 230.154,Z 460.429,A -85,B 0,C 180,E1 -19874.049,E2 -19874.049} C_VEL
LIN {X 0,Y 228.987,Z 465.669,A -85,B 0,C 180,E1 -19875.787,E2 -19875.787} C_VEL
LIN {X 0,Y 227.978,Z 470.037,A -85,B 0,C 180,E1 -19877.538,E2 -19877.538} C_VEL
LIN {X 0,Y 226.869,Z 475.188,A -85,B 0,C 180,E1 -19880.19,E2 -19880.19} C_VEL
LIN {X 0,Y 226.148,Z 478.967,A -85,B 0,C 180,E1 -19882.859,E2 -19882.859} C_VEL
LIN {X 0,Y 225.828,Z 480.833,A -85,B 0,C 180,E1 -19884.79,E2 -19884.79} C_VEL
LIN {X 0,Y 225.671,Z 481.94,A -85,B 0,C 180,E1 -19886.429,E2 -19886.429} C_VEL
LIN {X 0,Y 225.598,Z 482.71,A -85,B 0,C 180,E1 -19888.215,E2 -19888.215} C_VEL
LIN {X 0,Y 225.588,Z 483,A -85,B 0,C 180,E1 -19890,E2 -19890} C_VEL
LIN {X 0,Y 225.598,Z 482.701,A -85,B 0,C 180,E1 -19891.785,E2 -19891.785} C_VEL
LIN {X 0,Y 225.753,Z 480.985,A -85,B 0,C 180,E1 -19894.998,E2 -19894.998} C_VEL
LIN {X 0,Y 226.348,Z 477.757,A -85,B 0,C 180,E1 -19898.032,E2 -19898.032} C_VEL
LIN {X 0,Y 226.864,Z 475.111,A -85,B 0,C 180,E1 -19899.81,E2 -19899.81} C_VEL
LIN {X 0,Y 227.975,Z 469.938,A -85,B 0,C 180,E1 -19902.462,E2 -19902.462} C_VEL
LIN {X 0,Y 229.593,Z 463.114,A -85,B 0,C 180,E1 -19905.081,E2 -19905.081} C_VEL
LIN {X 0,Y 231.17,Z 455.654,A -85,B 0,C 180,E1 -19907.242,E2 -19907.242} C_VEL
LIN {X 0,Y 232.751,Z 448.295,A -85,B 0,C 180,E1 -19908.941,E2 -19908.941} C_VEL
LIN {X 0,Y 234.276,Z 440.409,A -85,B 0,C 180,E1 -19910.41,E2 -19910.41} C_VEL
LIN {X 0,Y 235.679,Z 432.071,A -85,B 0,C 180,E1 -19911.655,E2 -19911.655} C_VEL
LIN {X 0,Y 236.998,Z 422.207,A -85,B 0,C 180,E1 -19912.812,E2 -19912.812} C_VEL
LIN {X 0,Y 238.208,Z 410.636,A -85,B 0,C 180,E1 -19913.755,E2 -19913.755} C_VEL
LIN {X 0,Y 238.933,Z 401.354,A -85,B 0,C 180,E1 -19914.253,E2 -19914.253} C_VEL
LIN {X 0,Y 239.789,Z 374.459,A -85,B 0,C 180,E1 -19915.098,E2 -19915.098} C_VEL
LIN {X 0,Y 240.067,Z 362.378,A -85,B 0,C 180,E1 -19915.458,E2 -19915.458} C_VEL
LIN {X 0,Y 236.746,Z 342.688,A -85,B 0,C 180,E1 -19916.493,E2 -19916.493} C_VEL
LIN {X 0,Y 232.004,Z 330.255,A -85,B 0,C 180,E1 -19917.501,E2 -19917.501} C_VEL
LIN {X 0,Y 229.38,Z 323.84,A -85,B 0,C 180,E1 -19918.136,E2 -19918.136} C_VEL
LIN {X 0,Y 228.394,Z 319.234,A -85,B 0,C 180,E1 -19920.504,E2 -19920.504} C_VEL
LIN {X 0,Y 227.907,Z 316.989,A -85,B 0,C 180,E1 -19921.875,E2 -19921.875} C_VEL
LIN {X 0,Y 227.888,Z 316.907,A -85,B 0,C 180,E1 -19926.695,E2 -19926.695} C_VEL
LIN {X 0,Y 227.796,Z 316.895,A -85,B 0,C 180,E1 -19930.382,E2 -19930.382} C_VEL
LIN {X 0,Y 227.806,Z 316.922,A -85,B 0,C 180,E1 -19935.198,E2 -19935.198} C_VEL
LIN {X 0,Y 227.796,Z 316.883,A -85,B 0,C 180,E1 -19939.617,E2 -19939.617} C_VEL
LIN {X 0,Y 227.86,Z 316.901,A -85,B 0,C 180,E1 -19944.125,E2 -19944.125} C_VEL
LIN {X 0,Y 227.851,Z 316.911,A -85,B 0,C 180,E1 -19948.375,E2 -19948.375} C_VEL
LIN {X 0,Y 227.839,Z 316.913,A -85,B 0,C 180,E1 -19952.439,E2 -19952.439} C_VEL
LIN {X 0,Y 227.86,Z 316.903,A -85,B 0,C 180,E1 -19956.362,E2 -19956.362} C_VEL
LIN {X 0,Y 227.882,Z 316.906,A -85,B 0,C 180,E1 -19960.169,E2 -19960.169} C_VEL
LIN {X 0,Y 227.993,Z 316.892,A -85,B 0,C 180,E1 -19963.893,E2 -19963.893} C_VEL
LIN {X 0,Y 228.119,Z 316.878,A -85,B 0,C 180,E1 -19969.348,E2 -19969.348} C_VEL
LIN {X 0,Y 228.297,Z 316.851,A -85,B 0,C 180,E1 -19972.927,E2 -19972.927} C_VEL
LIN {X 0,Y 228.526,Z 316.827,A -85,B 0,C 180,E1 -19978.238,E2 -19978.238} C_VEL
LIN {X 0,Y 228.524,Z 316.828,A -85,B 0,C 180,E1 -19981.763,E2 -19981.763} C_VEL
LIN {X 0,Y 228.287,Z 316.853,A -85,B 0,C 180,E1 -19987.074,E2 -19987.074} C_VEL
LIN {X 0,Y 228.119,Z 316.878,A -85,B 0,C 180,E1 -19990.653,E2 -19990.653} C_VEL
LIN {X 0,Y 227.994,Z 316.891,A -85,B 0,C 180,E1 -19996.107,E2 -19996.107} C_VEL
LIN {X 0,Y 227.914,Z 316.89,A -85,B 0,C 180,E1 -20001.718,E2 -20001.718} C_VEL
LIN {X 0,Y 227.898,Z 316.909,A -85,B 0,C 180,E1 -20006.583,E2 -20006.583} C_VEL
LIN {X 0,Y 227.869,Z 316.9,A -85,B 0,C 180,E1 -20010.281,E2 -20010.281} C_VEL
LIN {X 0,Y 227.872,Z 316.912,A -85,B 0,C 180,E1 -20013.721,E2 -20013.721} C_VEL
LIN {X 0,Y 227.837,Z 316.875,A -85,B 0,C 180,E1 -20018.093,E2 -20018.093} C_VEL
LIN {X 0,Y 227.782,Z 316.916,A -85,B 0,C 180,E1 -20022.749,E2 -20022.749} C_VEL
LIN {X 0,Y 227.782,Z 316.901,A -85,B 0,C 180,E1 -20027.252,E2 -20027.252} C_VEL
LIN {X 0,Y 227.842,Z 316.916,A -85,B 0,C 180,E1 -20031.91,E2 -20031.91} C_VEL
LIN {X 0,Y 227.878,Z 316.901,A -85,B 0,C 180,E1 -20036.378,E2 -20036.378} C_VEL
LIN {X 0,Y 227.922,Z 317.015,A -85,B 0,C 180,E1 -20038.257,E2 -20038.257} C_VEL
LIN {X 0,Y 229.312,Z 323.719,A -85,B 0,C 180,E1 -20041.867,E2 -20041.867} C_VEL
LIN {X 0,Y 231.075,Z 328.199,A -85,B 0,C 180,E1 -20042.353,E2 -20042.353} C_VEL
LIN {X 0,Y 236.337,Z 341.411,A -85,B 0,C 180,E1 -20043.461,E2 -20043.461} C_VEL
LIN {X 0,Y 238.272,Z 351.029,A -85,B 0,C 180,E1 -20044.009,E2 -20044.009} C_VEL
LIN {X 0,Y 240.108,Z 363.407,A -85,B 0,C 180,E1 -20044.625,E2 -20044.625} C_VEL
LIN {X 0,Y 238.957,Z 399.979,A -85,B 0,C 180,E1 -20045.733,E2 -20045.733} C_VEL
LIN {X 0,Y 238.253,Z 409.934,A -85,B 0,C 180,E1 -20046.246,E2 -20046.246} C_VEL
LIN {X 0,Y 237.271,Z 420.539,A -85,B 0,C 180,E1 -20047.078,E2 -20047.078} C_VEL
LIN {X 0,Y 235.759,Z 431.777,A -85,B 0,C 180,E1 -20048.353,E2 -20048.353} C_VEL
LIN {X 0,Y 234.319,Z 440.168,A -85,B 0,C 180,E1 -20049.594,E2 -20049.594} C_VEL
LIN {X 0,Y 232.798,Z 448.094,A -85,B 0,C 180,E1 -20051.063,E2 -20051.063} C_VEL
LIN {X 0,Y 231.223,Z 455.486,A -85,B 0,C 180,E1 -20052.762,E2 -20052.762} C_VEL
LIN {X 0,Y 229.611,Z 462.976,A -85,B 0,C 180,E1 -20054.92,E2 -20054.92} C_VEL
LIN {X 0,Y 228.029,Z 469.843,A -85,B 0,C 180,E1 -20057.541,E2 -20057.541} C_VEL
LIN {X 0,Y 226.881,Z 475.035,A -85,B 0,C 180,E1 -20060.191,E2 -20060.191} C_VEL
LIN {X 0,Y 226.35,Z 477.7,A -85,B 0,C 180,E1 -20061.968,E2 -20061.968} C_VEL
LIN {X 0,Y 225.755,Z 480.943,A -85,B 0,C 180,E1 -20065.002,E2 -20065.002} C_VEL
LIN {X 0,Y 225.6,Z 482.693,A -85,B 0,C 180,E1 -20068.215,E2 -20068.215} C_VEL
LIN {X 0,Y 225.589,Z 482.999,A -85,B 0,C 180,E1 -20070,E2 -20070} C_VEL
LIN {X 0,Y 225.593,Z 482.718,A -85,B 0,C 180,E1 -20071.785,E2 -20071.785} C_VEL
LIN {X 0,Y 225.75,Z 481.081,A -85,B 0,C 180,E1 -20074.982,E2 -20074.982} C_VEL
LIN {X 0,Y 226.114,Z 479.024,A -85,B 0,C 180,E1 -20077.142,E2 -20077.142} C_VEL
LIN {X 0,Y 226.86,Z 475.264,A -85,B 0,C 180,E1 -20079.81,E2 -20079.81} C_VEL
LIN {X 0,Y 227.953,Z 470.132,A -85,B 0,C 180,E1 -20082.463,E2 -20082.463} C_VEL
LIN {X 0,Y 229.266,Z 464.613,A -85,B 0,C 180,E1 -20084.649,E2 -20084.649} C_VEL
LIN {X 0,Y 230.797,Z 457.678,A -85,B 0,C 180,E1 -20086.815,E2 -20086.815} C_VEL
LIN {X 0,Y 232.498,Z 449.717,A -85,B 0,C 180,E1 -20088.734,E2 -20088.734} C_VEL
LIN {X 0,Y 234.043,Z 442.127,A -85,B 0,C 180,E1 -20090.201,E2 -20090.201} C_VEL
LIN {X 0,Y 235.481,Z 434.171,A -85,B 0,C 180,E1 -20091.444,E2 -20091.444} C_VEL
LIN {X 0,Y 236.635,Z 425.949,A -85,B 0,C 180,E1 -20092.481,E2 -20092.481} C_VEL
LIN {X 0,Y 237.625,Z 418.029,A -85,B 0,C 180,E1 -20093.261,E2 -20093.261} C_VEL
LIN {X 0,Y 238.364,Z 409.349,A -85,B 0,C 180,E1 -20093.92,E2 -20093.92} C_VEL
LIN {X 0,Y 238.989,Z 400.183,A -85,B 0,C 180,E1 -20094.392,E2 -20094.392} C_VEL
LIN {X 0,Y 240.199,Z 362.867,A -85,B 0,C 180,E1 -20095.52,E2 -20095.52} C_VEL
LIN {X 0,Y 236.917,Z 343.096,A -85,B 0,C 180,E1 -20096.553,E2 -20096.553} C_VEL
LIN {X 0,Y 231.978,Z 330.168,A -85,B 0,C 180,E1 -20097.605,E2 -20097.605} C_VEL
LIN {X 0,Y 229.416,Z 323.948,A -85,B 0,C 180,E1 -20098.217,E2 -20098.217} C_VEL
LIN {X 0,Y 228.862,Z 321.366,A -85,B 0,C 180,E1 -20099.428,E2 -20099.428} C_VEL
LIN {X 0,Y 227.939,Z 316.978,A -85,B 0,C 180,E1 -20102,E2 -20102} C_VEL
LIN {X 0,Y 227.878,Z 316.907,A -85,B 0,C 180,E1 -20106.691,E2 -20106.691} C_VEL
LIN {X 0,Y 227.797,Z 316.896,A -85,B 0,C 180,E1 -20110.382,E2 -20110.382} C_VEL
LIN {X 0,Y 227.807,Z 316.921,A -85,B 0,C 180,E1 -20115.198,E2 -20115.198} C_VEL
LIN {X 0,Y 227.794,Z 316.885,A -85,B 0,C 180,E1 -20119.616,E2 -20119.616} C_VEL
LIN {X 0,Y 227.858,Z 316.899,A -85,B 0,C 180,E1 -20124.124,E2 -20124.124} C_VEL
LIN {X 0,Y 227.852,Z 316.912,A -85,B 0,C 180,E1 -20128.375,E2 -20128.375} C_VEL
LIN {X 0,Y 227.84,Z 316.912,A -85,B 0,C 180,E1 -20132.439,E2 -20132.439} C_VEL
LIN {X 0,Y 227.86,Z 316.904,A -85,B 0,C 180,E1 -20136.361,E2 -20136.361} C_VEL
LIN {X 0,Y 227.882,Z 316.905,A -85,B 0,C 180,E1 -20140.169,E2 -20140.169} C_VEL
LIN {X 0,Y 227.994,Z 316.892,A -85,B 0,C 180,E1 -20143.893,E2 -20143.893} C_VEL
LIN {X 0,Y 228.119,Z 316.878,A -85,B 0,C 180,E1 -20149.347,E2 -20149.347} C_VEL
LIN {X 0,Y 228.298,Z 316.852,A -85,B 0,C 180,E1 -20152.927,E2 -20152.927} C_VEL
LIN {X 0,Y 228.526,Z 316.827,A -85,B 0,C 180,E1 -20158.237,E2 -20158.237} C_VEL
LIN {X 0,Y 228.524,Z 316.828,A -85,B 0,C 180,E1 -20161.762,E2 -20161.762} C_VEL
LIN {X 0,Y 228.286,Z 316.853,A -85,B 0,C 180,E1 -20167.073,E2 -20167.073} C_VEL
LIN {X 0,Y 228.119,Z 316.878,A -85,B 0,C 180,E1 -20170.652,E2 -20170.652} C_VEL
LIN {X 0,Y 227.993,Z 316.892,A -85,B 0,C 180,E1 -20176.107,E2 -20176.107} C_VEL
LIN {X 0,Y 227.913,Z 316.89,A -85,B 0,C 180,E1 -20181.718,E2 -20181.718} C_VEL
LIN {X 0,Y 227.898,Z 316.909,A -85,B 0,C 180,E1 -20186.582,E2 -20186.582} C_VEL
LIN {X 0,Y 227.868,Z 316.901,A -85,B 0,C 180,E1 -20190.28,E2 -20190.28} C_VEL
LIN {X 0,Y 227.871,Z 316.912,A -85,B 0,C 180,E1 -20193.721,E2 -20193.721} C_VEL
LIN {X 0,Y 227.86,Z 316.899,A -85,B 0,C 180,E1 -20195.944,E2 -20195.944} C_VEL
LIN {X 0,Y 227.18,Z 316.966,A -85,B 0,C 180,E1 -20197.419,E2 -20197.419} C_VEL
LIN {X 0,Y 224.285,Z 317.328,A -85,B 0,C 180,E1 -20199.823,E2 -20199.823} C_VEL
LIN {X 0,Y 221.835,Z 317.646,A -85,B 0,C 180,E1 -20201.785,E2 -20201.785} C_VEL
LIN {X 0,Y 220.801,Z 317.792,A -85,B 0,C 180,E1 -20203.31,E2 -20203.31} C_VEL
LIN {X 0,Y 220.726,Z 317.799,A -85,B 0,C 180,E1 -20203.827,E2 -20203.827} C_VEL
LIN {X 0,Y 220.744,Z 317.768,A -85,B 0,C 180,E1 -20208.043,E2 -20208.043} C_VEL
LIN {X 0,Y 220.822,Z 317.789,A -85,B 0,C 180,E1 -20212.794,E2 -20212.794} C_VEL
LIN {X 0,Y 220.887,Z 317.894,A -85,B 0,C 180,E1 -20217.499,E2 -20217.499} C_VEL
LIN {X 0,Y 222.113,Z 323.669,A -85,B 0,C 180,E1 -20220.764,E2 -20220.764} C_VEL
LIN {X 0,Y 223.801,Z 327.682,A -85,B 0,C 180,E1 -20221.251,E2 -20221.251} C_VEL
LIN {X 0,Y 230.58,Z 344.575,A -85,B 0,C 180,E1 -20222.754,E2 -20222.754} C_VEL
LIN {X 0,Y 233.415,Z 361.529,A -85,B 0,C 180,E1 -20223.683,E2 -20223.683} C_VEL
LIN {X 0,Y 233.741,Z 366.749,A -85,B 0,C 180,E1 -20223.898,E2 -20223.898} C_VEL
LIN {X 0,Y 232.608,Z 400.236,A -85,B 0,C 180,E1 -20224.942,E2 -20224.942} C_VEL
LIN {X 0,Y 231.903,Z 409.705,A -85,B 0,C 180,E1 -20225.441,E2 -20225.441} C_VEL
LIN {X 0,Y 230.772,Z 420.512,A -85,B 0,C 180,E1 -20226.296,E2 -20226.296} C_VEL
LIN {X 0,Y 229.368,Z 430.881,A -85,B 0,C 180,E1 -20227.48,E2 -20227.48} C_VEL
LIN {X 0,Y 227.889,Z 439.432,A -85,B 0,C 180,E1 -20228.755,E2 -20228.755} C_VEL
LIN {X 0,Y 226.237,Z 447.478,A -85,B 0,C 180,E1 -20230.256,E2 -20230.256} C_VEL
LIN {X 0,Y 224.793,Z 454.124,A -85,B 0,C 180,E1 -20231.782,E2 -20231.782} C_VEL
LIN {X 0,Y 223.323,Z 460.431,A -85,B 0,C 180,E1 -20233.547,E2 -20233.547} C_VEL
LIN {X 0,Y 222.121,Z 465.671,A -85,B 0,C 180,E1 -20235.338,E2 -20235.338} C_VEL
LIN {X 0,Y 221.042,Z 470.039,A -85,B 0,C 180,E1 -20237.141,E2 -20237.141} C_VEL
LIN {X 0,Y 219.879,Z 475.189,A -85,B 0,C 180,E1 -20239.875,E2 -20239.875} C_VEL
LIN {X 0,Y 219.11,Z 478.968,A -85,B 0,C 180,E1 -20242.629,E2 -20242.629} C_VEL
LIN {X 0,Y 218.721,Z 481.108,A -85,B 0,C 180,E1 -20244.935,E2 -20244.935} C_VEL
LIN {X 0,Y 218.503,Z 482.71,A -85,B 0,C 180,E1 -20248.157,E2 -20248.157} C_VEL
LIN {X 0,Y 218.49,Z 483,A -85,B 0,C 180,E1 -20250,E2 -20250} C_VEL
LIN {X 0,Y 218.503,Z 482.701,A -85,B 0,C 180,E1 -20251.843,E2 -20251.843} C_VEL
LIN {X 0,Y 218.652,Z 481.244,A -85,B 0,C 180,E1 -20254.857,E2 -20254.857} C_VEL
LIN {X 0,Y 219.065,Z 478.907,A -85,B 0,C 180,E1 -20257.373,E2 -20257.373} C_VEL
LIN {X 0,Y 219.874,Z 475.11,A -85,B 0,C 180,E1 -20260.125,E2 -20260.125} C_VEL
LIN {X 0,Y 221.039,Z 469.937,A -85,B 0,C 180,E1 -20262.86,E2 -20262.86} C_VEL
LIN {X 0,Y 222.745,Z 463.112,A -85,B 0,C 180,E1 -20265.556,E2 -20265.556} C_VEL
LIN {X 0,Y 224.391,Z 455.651,A -85,B 0,C 180,E1 -20267.78,E2 -20267.78} C_VEL
LIN {X 0,Y 226.054,Z 448.292,A -85,B 0,C 180,E1 -20269.524,E2 -20269.524} C_VEL
LIN {X 0,Y 227.65,Z 440.406,A -85,B 0,C 180,E1 -20271.031,E2 -20271.031} C_VEL
LIN {X 0,Y 229.098,Z 432.067,A -85,B 0,C 180,E1 -20272.31,E2 -20272.31} C_VEL
LIN {X 0,Y 230.596,Z 421.41,A -85,B 0,C 180,E1 -20273.577,E2 -20273.577} C_VEL
LIN {X 0,Y 231.837,Z 409.815,A -85,B 0,C 180,E1 -20274.508,E2 -20274.508} C_VEL
LIN {X 0,Y 232.508,Z 400.716,A -85,B 0,C 180,E1 -20274.997,E2 -20274.997} C_VEL
LIN {X 0,Y 233.693,Z 363.479,A -85,B 0,C 180,E1 -20276.167,E2 -20276.167} C_VEL
LIN {X 0,Y 230.52,Z 344.715,A -85,B 0,C 180,E1 -20277.196,E2 -20277.196} C_VEL
LIN {X 0,Y 225.598,Z 331.996,A -85,B 0,C 180,E1 -20278.289,E2 -20278.289} C_VEL
LIN {X 0,Y 222.173,Z 323.887,A -85,B 0,C 180,E1 -20279.123,E2 -20279.123} C_VEL
LIN {X 0,Y 221.367,Z 320.305,A -85,B 0,C 180,E1 -20280.997,E2 -20280.997} C_VEL
LIN {X 0,Y 220.883,Z 317.879,A -85,B 0,C 180,E1 -20282.499,E2 -20282.499} C_VEL
LIN {X 0,Y 220.807,Z 317.792,A -85,B 0,C 180,E1 -20287.277,E2 -20287.277} C_VEL
LIN {X 0,Y 220.744,Z 317.769,A -85,B 0,C 180,E1 -20291.957,E2 -20291.957} C_VEL
LIN {X 0,Y 220.749,Z 317.801,A -85,B 0,C 180,E1 -20295.54,E2 -20295.54} C_VEL
LIN {X 0,Y 220.777,Z 317.748,A -85,B 0,C 180,E1 -20300.457,E2 -20300.457} C_VEL
LIN {X 0,Y 220.821,Z 317.757,A -85,B 0,C 180,E1 -20302.793,E2 -20302.793} C_VEL
LIN {X 0,Y 220.807,Z 317.792,A -85,B 0,C 180,E1 -20307.243,E2 -20307.243} C_VEL
LIN {X 0,Y 220.794,Z 317.785,A -85,B 0,C 180,E1 -20311.481,E2 -20311.481} C_VEL
LIN {X 0,Y 220.798,Z 317.789,A -85,B 0,C 180,E1 -20315.557,E2 -20315.557} C_VEL
LIN {X 0,Y 220.84,Z 317.781,A -85,B 0,C 180,E1 -20319.509,E2 -20319.509} C_VEL
LIN {X 0,Y 220.96,Z 317.77,A -85,B 0,C 180,E1 -20323.366,E2 -20323.366} C_VEL
LIN {X 0,Y 221.044,Z 317.759,A -85,B 0,C 180,E1 -20329.003,E2 -20329.003} C_VEL
LIN {X 0,Y 221.235,Z 317.732,A -85,B 0,C 180,E1 -20332.7,E2 -20332.7} C_VEL
LIN {X 0,Y 221.46,Z 317.706,A -85,B 0,C 180,E1 -20338.182,E2 -20338.182} C_VEL
LIN {X 0,Y 221.457,Z 317.707,A -85,B 0,C 180,E1 -20341.819,E2 -20341.819} C_VEL
LIN {X 0,Y 221.224,Z 317.733,A -85,B 0,C 180,E1 -20347.301,E2 -20347.301} C_VEL
LIN {X 0,Y 221.044,Z 317.759,A -85,B 0,C 180,E1 -20350.998,E2 -20350.998} C_VEL
LIN {X 0,Y 220.961,Z 317.769,A -85,B 0,C 180,E1 -20356.634,E2 -20356.634} C_VEL
LIN {X 0,Y 220.841,Z 317.781,A -85,B 0,C 180,E1 -20360.491,E2 -20360.491} C_VEL
LIN {X 0,Y 220.798,Z 317.789,A -85,B 0,C 180,E1 -20364.443,E2 -20364.443} C_VEL
LIN {X 0,Y 220.794,Z 317.786,A -85,B 0,C 180,E1 -20368.52,E2 -20368.52} C_VEL
LIN {X 0,Y 220.808,Z 317.792,A -85,B 0,C 180,E1 -20372.758,E2 -20372.758} C_VEL
LIN {X 0,Y 220.798,Z 317.759,A -85,B 0,C 180,E1 -20377.276,E2 -20377.276} C_VEL
LIN {X 0,Y 220.745,Z 317.781,A -85,B 0,C 180,E1 -20381.959,E2 -20381.959} C_VEL
LIN {X 0,Y 220.75,Z 317.796,A -85,B 0,C 180,E1 -20385.541,E2 -20385.541} C_VEL
LIN {X 0,Y 220.779,Z 317.776,A -85,B 0,C 180,E1 -20390.458,E2 -20390.458} C_VEL
LIN {X 0,Y 220.824,Z 317.79,A -85,B 0,C 180,E1 -20392.794,E2 -20392.794} C_VEL
LIN {X 0,Y 220.895,Z 317.918,A -85,B 0,C 180,E1 -20397.628,E2 -20397.628} C_VEL
LIN {X 0,Y 222.085,Z 323.716,A -85,B 0,C 180,E1 -20400.863,E2 -20400.863} C_VEL
LIN {X 0,Y 223.614,Z 327.39,A -85,B 0,C 180,E1 -20401.317,E2 -20401.317} C_VEL
LIN {X 0,Y 229.969,Z 342.912,A -85,B 0,C 180,E1 -20402.716,E2 -20402.716} C_VEL
LIN {X 0,Y 231.455,Z 349.181,A -85,B 0,C 180,E1 -20403.12,E2 -20403.12} C_VEL
LIN {X 0,Y 233.708,Z 364.312,A -85,B 0,C 180,E1 -20403.908,E2 -20403.908} C_VEL
LIN {X 0,Y 232.508,Z 400.387,A -85,B 0,C 180,E1 -20405.033,E2 -20405.033} C_VEL
LIN {X 0,Y 231.743,Z 410.464,A -85,B 0,C 180,E1 -20405.573,E2 -20405.573} C_VEL
LIN {X 0,Y 230.541,Z 421.945,A -85,B 0,C 180,E1 -20406.525,E2 -20406.525} C_VEL
LIN {X 0,Y 229.185,Z 431.782,A -85,B 0,C 180,E1 -20407.699,E2 -20407.699} C_VEL
LIN {X 0,Y 227.693,Z 440.172,A -85,B 0,C 180,E1 -20408.973,E2 -20408.973} C_VEL
LIN {X 0,Y 226.107,Z 448.097,A -85,B 0,C 180,E1 -20410.48,E2 -20410.48} C_VEL
LIN {X 0,Y 224.437,Z 455.489,A -85,B 0,C 180,E1 -20412.224,E2 -20412.224} C_VEL
LIN {X 0,Y 222.765,Z 462.978,A -85,B 0,C 180,E1 -20414.445,E2 -20414.445} C_VEL
LIN {X 0,Y 221.084,Z 469.844,A -85,B 0,C 180,E1 -20417.143,E2 -20417.143} C_VEL
LIN {X 0,Y 219.895,Z 475.037,A -85,B 0,C 180,E1 -20419.876,E2 -20419.876} C_VEL
LIN {X 0,Y 219.306,Z 477.701,A -85,B 0,C 180,E1 -20421.709,E2 -20421.709} C_VEL
LIN {X 0,Y 218.741,Z 480.619,A -85,B 0,C 180,E1 -20424.469,E2 -20424.469} C_VEL
LIN {X 0,Y 218.586,Z 481.892,A -85,B 0,C 180,E1 -20426.313,E2 -20426.313} C_VEL
LIN {X 0,Y 218.505,Z 482.693,A -85,B 0,C 180,E1 -20428.157,E2 -20428.157} C_VEL
LIN {X 0,Y 218.491,Z 482.999,A -85,B 0,C 180,E1 -20430,E2 -20430} C_VEL
LIN {X 0,Y 218.497,Z 482.717,A -85,B 0,C 180,E1 -20431.843,E2 -20431.843} C_VEL
LIN {X 0,Y 218.644,Z 481.338,A -85,B 0,C 180,E1 -20434.826,E2 -20434.826} C_VEL
LIN {X 0,Y 219.066,Z 479.023,A -85,B 0,C 180,E1 -20437.373,E2 -20437.373} C_VEL
LIN {X 0,Y 219.87,Z 475.262,A -85,B 0,C 180,E1 -20440.125,E2 -20440.125} C_VEL
LIN {X 0,Y 221.025,Z 470.131,A -85,B 0,C 180,E1 -20442.86,E2 -20442.86} C_VEL
LIN {X 0,Y 222.416,Z 464.611,A -85,B 0,C 180,E1 -20445.11,E2 -20445.11} C_VEL
LIN {X 0,Y 224.009,Z 457.675,A -85,B 0,C 180,E1 -20447.34,E2 -20447.34} C_VEL
LIN {X 0,Y 225.79,Z 449.714,A -85,B 0,C 180,E1 -20449.312,E2 -20449.312} C_VEL
LIN {X 0,Y 227.412,Z 442.123,A -85,B 0,C 180,E1 -20450.817,E2 -20450.817} C_VEL
LIN {X 0,Y 228.894,Z 434.166,A -85,B 0,C 180,E1 -20452.093,E2 -20452.093} C_VEL
LIN {X 0,Y 229.825,Z 427.815,A -85,B 0,C 180,E1 -20452.947,E2 -20452.947} C_VEL
LIN {X 0,Y 231.16,Z 417.565,A -85,B 0,C 180,E1 -20453.997,E2 -20453.997} C_VEL
LIN {X 0,Y 231.936,Z 409.019,A -85,B 0,C 180,E1 -20454.649,E2 -20454.649} C_VEL
LIN {X 0,Y 232.588,Z 399.517,A -85,B 0,C 180,E1 -20455.139,E2 -20455.139} C_VEL
LIN {X 0,Y 233.682,Z 363.082,A -85,B 0,C 180,E1 -20456.277,E2 -20456.277} C_VEL
LIN {X 0,Y 230.764,Z 345.307,A -85,B 0,C 180,E1 -20457.243,E2 -20457.243} C_VEL
LIN {X 0,Y 226.099,Z 333.22,A -85,B 0,C 180,E1 -20458.279,E2 -20458.279} C_VEL
LIN {X 0,Y 222.159,Z 323.861,A -85,B 0,C 180,E1 -20459.236,E2 -20459.236} C_VEL
LIN {X 0,Y 221.45,Z 320.412,A -85,B 0,C 180,E1 -20461.032,E2 -20461.032} C_VEL
LIN {X 0,Y 220.906,Z 317.872,A -85,B 0,C 180,E1 -20462.62,E2 -20462.62} C_VEL
LIN {X 0,Y 220.8,Z 317.792,A -85,B 0,C 180,E1 -20467.274,E2 -20467.274} C_VEL
LIN {X 0,Y 220.745,Z 317.768,A -85,B 0,C 180,E1 -20471.957,E2 -20471.957} C_VEL
LIN {X 0,Y 220.75,Z 317.802,A -85,B 0,C 180,E1 -20475.54,E2 -20475.54} C_VEL
LIN {X 0,Y 220.776,Z 317.749,A -85,B 0,C 180,E1 -20480.456,E2 -20480.456} C_VEL
LIN {X 0,Y 220.822,Z 317.755,A -85,B 0,C 180,E1 -20482.792,E2 -20482.792} C_VEL
LIN {X 0,Y 220.808,Z 317.793,A -85,B 0,C 180,E1 -20487.242,E2 -20487.242} C_VEL
LIN {X 0,Y 220.794,Z 317.784,A -85,B 0,C 180,E1 -20491.48,E2 -20491.48} C_VEL
LIN {X 0,Y 220.798,Z 317.79,A -85,B 0,C 180,E1 -20495.557,E2 -20495.557} C_VEL
LIN {X 0,Y 220.841,Z 317.78,A -85,B 0,C 180,E1 -20499.509,E2 -20499.509} C_VEL
LIN {X 0,Y 220.961,Z 317.77,A -85,B 0,C 180,E1 -20503.366,E2 -20503.366} C_VEL
LIN {X 0,Y 221.044,Z 317.759,A -85,B 0,C 180,E1 -20509.002,E2 -20509.002} C_VEL
LIN {X 0,Y 221.235,Z 317.732,A -85,B 0,C 180,E1 -20512.7,E2 -20512.7} C_VEL
LIN {X 0,Y 221.46,Z 317.706,A -85,B 0,C 180,E1 -20518.181,E2 -20518.181} C_VEL
LIN {X 0,Y 221.457,Z 317.707,A -85,B 0,C 180,E1 -20521.818,E2 -20521.818} C_VEL
LIN {X 0,Y 221.224,Z 317.733,A -85,B 0,C 180,E1 -20527.3,E2 -20527.3} C_VEL
LIN {X 0,Y 221.044,Z 317.759,A -85,B 0,C 180,E1 -20530.997,E2 -20530.997} C_VEL
LIN {X 0,Y 220.96,Z 317.77,A -85,B 0,C 180,E1 -20536.634,E2 -20536.634} C_VEL
LIN {X 0,Y 220.84,Z 317.78,A -85,B 0,C 180,E1 -20540.491,E2 -20540.491} C_VEL
LIN {X 0,Y 220.798,Z 317.79,A -85,B 0,C 180,E1 -20544.443,E2 -20544.443} C_VEL
LIN {X 0,Y 220.794,Z 317.785,A -85,B 0,C 180,E1 -20548.519,E2 -20548.519} C_VEL
LIN {X 0,Y 220.807,Z 317.793,A -85,B 0,C 180,E1 -20552.757,E2 -20552.757} C_VEL
LIN {X 0,Y 220.797,Z 317.757,A -85,B 0,C 180,E1 -20557.275,E2 -20557.275} C_VEL
LIN {X 0,Y 220.744,Z 317.783,A -85,B 0,C 180,E1 -20561.958,E2 -20561.958} C_VEL
LIN {X 0,Y 220.726,Z 317.799,A -85,B 0,C 180,E1 -20563.827,E2 -20563.827} C_VEL
LIN {X 0,Y 220.074,Z 317.884,A -85,B 0,C 180,E1 -20565.351,E2 -20565.351} C_VEL
LIN {X 0,Y 217.21,Z 318.234,A -85,B 0,C 180,E1 -20567.839,E2 -20567.839} C_VEL
LIN {X 0,Y 214.785,Z 318.532,A -85,B 0,C 180,E1 -20569.871,E2 -20569.871} C_VEL
LIN {X 0,Y 213.775,Z 318.664,A -85,B 0,C 180,E1 -20571.449,E2 -20571.449} C_VEL
LIN {X 0,Y 213.71,Z 318.676,A -85,B 0,C 180,E1 -20571.984,E2 -20571.984} C_VEL
LIN {X 0,Y 213.81,Z 318.791,A -85,B 0,C 180,E1 -20576.806,E2 -20576.806} C_VEL
LIN {X 0,Y 214.923,Z 323.764,A -85,B 0,C 180,E1 -20579.704,E2 -20579.704} C_VEL
LIN {X 0,Y 217.311,Z 329.362,A -85,B 0,C 180,E1 -20580.37,E2 -20580.37} C_VEL
LIN {X 0,Y 223.73,Z 344.839,A -85,B 0,C 180,E1 -20581.855,E2 -20581.855} C_VEL
LIN {X 0,Y 224.979,Z 349.303,A -85,B 0,C 180,E1 -20582.183,E2 -20582.183} C_VEL
LIN {X 0,Y 227.338,Z 364.493,A -85,B 0,C 180,E1 -20583.025,E2 -20583.025} C_VEL
LIN {X 0,Y 226.212,Z 400.071,A -85,B 0,C 180,E1 -20584.173,E2 -20584.173} C_VEL
LIN {X 0,Y 225.474,Z 409.707,A -85,B 0,C 180,E1 -20584.692,E2 -20584.692} C_VEL
LIN {X 0,Y 224.229,Z 420.977,A -85,B 0,C 180,E1 -20585.609,E2 -20585.609} C_VEL
LIN {X 0,Y 222.84,Z 430.885,A -85,B 0,C 180,E1 -20586.783,E2 -20586.783} C_VEL
LIN {X 0,Y 221.28,Z 439.436,A -85,B 0,C 180,E1 -20588.088,E2 -20588.088} C_VEL
LIN {X 0,Y 219.58,Z 447.481,A -85,B 0,C 180,E1 -20589.631,E2 -20589.631} C_VEL
LIN {X 0,Y 218.066,Z 454.126,A -85,B 0,C 180,E1 -20591.199,E2 -20591.199} C_VEL
LIN {X 0,Y 216.511,Z 460.434,A -85,B 0,C 180,E1 -20593.014,E2 -20593.014} C_VEL
LIN {X 0,Y 215.255,Z 465.673,A -85,B 0,C 180,E1 -20594.859,E2 -20594.859} C_VEL
LIN {X 0,Y 214.129,Z 470.04,A -85,B 0,C 180,E1 -20596.718,E2 -20596.718} C_VEL
LIN {X 0,Y 212.881,Z 475.19,A -85,B 0,C 180,E1 -20599.539,E2 -20599.539} C_VEL
LIN {X 0,Y 212.068,Z 478.968,A -85,B 0,C 180,E1 -20602.383,E2 -20602.383} C_VEL
LIN {X 0,Y 211.617,Z 481.358,A -85,B 0,C 180,E1 -20605.087,E2 -20605.087} C_VEL
LIN {X 0,Y 211.411,Z 482.71,A -85,B 0,C 180,E1 -20608.095,E2 -20608.095} C_VEL
LIN {X 0,Y 211.394,Z 483,A -85,B 0,C 180,E1 -20610,E2 -20610} C_VEL
LIN {X 0,Y 211.411,Z 482.701,A -85,B 0,C 180,E1 -20611.905,E2 -20611.905} C_VEL
LIN {X 0,Y 211.541,Z 481.478,A -85,B 0,C 180,E1 -20614.669,E2 -20614.669} C_VEL
LIN {X 0,Y 212.015,Z 478.906,A -85,B 0,C 180,E1 -20617.619,E2 -20617.619} C_VEL
LIN {X 0,Y 212.875,Z 475.109,A -85,B 0,C 180,E1 -20620.462,E2 -20620.462} C_VEL
LIN {X 0,Y 214.127,Z 469.935,A -85,B 0,C 180,E1 -20623.282,E2 -20623.282} C_VEL
LIN {X 0,Y 215.886,Z 463.109,A -85,B 0,C 180,E1 -20626.064,E2 -20626.064} C_VEL
LIN {X 0,Y 217.64,Z 455.649,A -85,B 0,C 180,E1 -20628.351,E2 -20628.351} C_VEL
LIN {X 0,Y 219.384,Z 448.288,A -85,B 0,C 180,E1 -20630.143,E2 -20630.143} C_VEL
LIN {X 0,Y 221.05,Z 440.402,A -85,B 0,C 180,E1 -20631.69,E2 -20631.69} C_VEL
LIN {X 0,Y 222.553,Z 432.062,A -85,B 0,C 180,E1 -20633.003,E2 -20633.003} C_VEL
LIN {X 0,Y 224.08,Z 421.682,A -85,B 0,C 180,E1 -20634.273,E2 -20634.273} C_VEL
LIN {X 0,Y 225.354,Z 410.229,A -85,B 0,C 180,E1 -20635.231,E2 -20635.231} C_VEL
LIN {X 0,Y 226.092,Z 400.833,A -85,B 0,C 180,E1 -20635.751,E2 -20635.751} C_VEL
LIN {X 0,Y 227.339,Z 364.664,A -85,B 0,C 180,E1 -20636.914,E2 -20636.914} C_VEL
LIN {X 0,Y 224.466,Z 347.127,A -85,B 0,C 180,E1 -20637.907,E2 -20637.907} C_VEL
LIN {X 0,Y 218.929,Z 333.024,A -85,B 0,C 180,E1 -20639.194,E2 -20639.194} C_VEL
LIN {X 0,Y 214.976,Z 323.987,A -85,B 0,C 180,E1 -20640.181,E2 -20640.181} C_VEL
LIN {X 0,Y 214.327,Z 321.169,A -85,B 0,C 180,E1 -20641.644,E2 -20641.644} C_VEL
LIN {X 0,Y 213.807,Z 318.735,A -85,B 0,C 180,E1 -20643.265,E2 -20643.265} C_VEL
LIN {X 0,Y 213.721,Z 318.676,A -85,B 0,C 180,E1 -20647.888,E2 -20647.888} C_VEL
LIN {X 0,Y 213.694,Z 318.644,A -85,B 0,C 180,E1 -20651.128,E2 -20651.128} C_VEL
LIN {X 0,Y 213.698,Z 318.663,A -85,B 0,C 180,E1 -20653.679,E2 -20653.679} C_VEL
LIN {X 0,Y 213.698,Z 318.679,A -85,B 0,C 180,E1 -20656.345,E2 -20656.345} C_VEL
LIN {X 0,Y 213.699,Z 318.627,A -85,B 0,C 180,E1 -20661.328,E2 -20661.328} C_VEL
LIN {X 0,Y 213.75,Z 318.67,A -85,B 0,C 180,E1 -20666.017,E2 -20666.017} C_VEL
LIN {X 0,Y 213.743,Z 318.656,A -85,B 0,C 180,E1 -20670.449,E2 -20670.449} C_VEL
LIN {X 0,Y 213.746,Z 318.671,A -85,B 0,C 180,E1 -20674.695,E2 -20674.695} C_VEL
LIN {X 0,Y 213.769,Z 318.653,A -85,B 0,C 180,E1 -20678.799,E2 -20678.799} C_VEL
LIN {X 0,Y 213.873,Z 318.654,A -85,B 0,C 180,E1 -20682.798,E2 -20682.798} C_VEL
LIN {X 0,Y 213.904,Z 318.631,A -85,B 0,C 180,E1 -20686.704,E2 -20686.704} C_VEL
LIN {X 0,Y 214.128,Z 318.624,A -85,B 0,C 180,E1 -20690.555,E2 -20690.555} C_VEL
LIN {X 0,Y 214.066,Z 318.61,A -85,B 0,C 180,E1 -20694.348,E2 -20694.348} C_VEL
LIN {X 0,Y 214.396,Z 318.585,A -85,B 0,C 180,E1 -20698.122,E2 -20698.122} C_VEL
LIN {X 0,Y 214.505,Z 318.58,A -85,B 0,C 180,E1 -20700,E2 -20700} C_VEL
LIN {X 0,Y 214.394,Z 318.586,A -85,B 0,C 180,E1 -20701.879,E2 -20701.879} C_VEL
LIN {X 0,Y 214.166,Z 318.613,A -85,B 0,C 180,E1 -20707.543,E2 -20707.543} C_VEL
LIN {X 0,Y 213.976,Z 318.636,A -85,B 0,C 180,E1 -20711.366,E2 -20711.366} C_VEL
LIN {X 0,Y 213.86,Z 318.643,A -85,B 0,C 180,E1 -20715.243,E2 -20715.243} C_VEL
LIN {X 0,Y 213.785,Z 318.667,A -85,B 0,C 180,E1 -20719.193,E2 -20719.193} C_VEL
LIN {X 0,Y 213.78,Z 318.651,A -85,B 0,C 180,E1 -20723.235,E2 -20723.235} C_VEL
LIN {X 0,Y 213.781,Z 318.664,A -85,B 0,C 180,E1 -20727.427,E2 -20727.427} C_VEL
LIN {X 0,Y 213.755,Z 318.667,A -85,B 0,C 180,E1 -20731.74,E2 -20731.74} C_VEL
LIN {X 0,Y 213.738,Z 318.65,A -85,B 0,C 180,E1 -20736.29,E2 -20736.29} C_VEL
LIN {X 0,Y 213.695,Z 318.643,A -85,B 0,C 180,E1 -20741.13,E2 -20741.13} C_VEL
LIN {X 0,Y 213.699,Z 318.679,A -85,B 0,C 180,E1 -20743.681,E2 -20743.681} C_VEL
LIN {X 0,Y 213.699,Z 318.663,A -85,B 0,C 180,E1 -20746.346,E2 -20746.346} C_VEL
LIN {X 0,Y 213.706,Z 318.669,A -85,B 0,C 180,E1 -20751.331,E2 -20751.331} C_VEL
LIN {X 0,Y 213.763,Z 318.653,A -85,B 0,C 180,E1 -20756.02,E2 -20756.02} C_VEL
LIN {X 0,Y 213.874,Z 318.91,A -85,B 0,C 180,E1 -20757.027,E2 -20757.027} C_VEL
LIN {X 0,Y 214.901,Z 323.834,A -85,B 0,C 180,E1 -20759.823,E2 -20759.823} C_VEL
LIN {X 0,Y 217.817,Z 330.545,A -85,B 0,C 180,E1 -20760.596,E2 -20760.596} C_VEL
LIN {X 0,Y 223.995,Z 345.588,A -85,B 0,C 180,E1 -20762.02,E2 -20762.02} C_VEL
LIN {X 0,Y 225.294,Z 351.222,A -85,B 0,C 180,E1 -20762.394,E2 -20762.394} C_VEL
LIN {X 0,Y 227.29,Z 364.272,A -85,B 0,C 180,E1 -20763.111,E2 -20763.111} C_VEL
LIN {X 0,Y 226.099,Z 400.41,A -85,B 0,C 180,E1 -20764.274,E2 -20764.274} C_VEL
LIN {X 0,Y 225.259,Z 411.002,A -85,B 0,C 180,E1 -20764.861,E2 -20764.861} C_VEL
LIN {X 0,Y 223.909,Z 422.976,A -85,B 0,C 180,E1 -20765.919,E2 -20765.919} C_VEL
LIN {X 0,Y 222.63,Z 431.787,A -85,B 0,C 180,E1 -20767.005,E2 -20767.005} C_VEL
LIN {X 0,Y 221.092,Z 440.176,A -85,B 0,C 180,E1 -20768.314,E2 -20768.314} C_VEL
LIN {X 0,Y 219.433,Z 448.1,A -85,B 0,C 180,E1 -20769.861,E2 -20769.861} C_VEL
LIN {X 0,Y 217.681,Z 455.492,A -85,B 0,C 180,E1 -20771.653,E2 -20771.653} C_VEL
LIN {X 0,Y 215.909,Z 462.981,A -85,B 0,C 180,E1 -20773.938,E2 -20773.938} C_VEL
LIN {X 0,Y 214.164,Z 469.846,A -85,B 0,C 180,E1 -20776.72,E2 -20776.72} C_VEL
LIN {X 0,Y 212.899,Z 475.038,A -85,B 0,C 180,E1 -20779.54,E2 -20779.54} C_VEL
LIN {X 0,Y 212.288,Z 477.702,A -85,B 0,C 180,E1 -20781.433,E2 -20781.433} C_VEL
LIN {X 0,Y 211.663,Z 480.619,A -85,B 0,C 180,E1 -20784.283,E2 -20784.283} C_VEL
LIN {X 0,Y 211.49,Z 481.892,A -85,B 0,C 180,E1 -20786.189,E2 -20786.189} C_VEL
LIN {X 0,Y 211.413,Z 482.693,A -85,B 0,C 180,E1 -20788.095,E2 -20788.095} C_VEL
LIN {X 0,Y 211.395,Z 482.999,A -85,B 0,C 180,E1 -20790,E2 -20790} C_VEL
LIN {X 0,Y 211.405,Z 482.717,A -85,B 0,C 180,E1 -20791.905,E2 -20791.905} C_VEL
LIN {X 0,Y 211.536,Z 481.542,A -85,B 0,C 180,E1 -20794.645,E2 -20794.645} C_VEL
LIN {X 0,Y 212.016,Z 479.022,A -85,B 0,C 180,E1 -20797.619,E2 -20797.619} C_VEL
LIN {X 0,Y 212.871,Z 475.261,A -85,B 0,C 180,E1 -20800.462,E2 -20800.462} C_VEL
LIN {X 0,Y 214.101,Z 470.129,A -85,B 0,C 180,E1 -20803.284,E2 -20803.284} C_VEL
LIN {X 0,Y 215.556,Z 464.609,A -85,B 0,C 180,E1 -20805.603,E2 -20805.603} C_VEL
LIN {X 0,Y 217.24,Z 457.673,A -85,B 0,C 180,E1 -20807.898,E2 -20807.898} C_VEL
LIN {X 0,Y 219.109,Z 449.71,A -85,B 0,C 180,E1 -20809.925,E2 -20809.925} C_VEL
LIN {X 0,Y 220.794,Z 442.119,A -85,B 0,C 180,E1 -20811.472,E2 -20811.472} C_VEL
LIN {X 0,Y 222.335,Z 434.161,A -85,B 0,C 180,E1 -20812.781,E2 -20812.781} C_VEL
LIN {X 0,Y 223.322,Z 427.809,A -85,B 0,C 180,E1 -20813.655,E2 -20813.655} C_VEL
LIN {X 0,Y 224.552,Z 418.914,A -85,B 0,C 180,E1 -20814.611,E2 -20814.611} C_VEL
LIN {X 0,Y 225.443,Z 409.708,A -85,B 0,C 180,E1 -20815.357,E2 -20815.357} C_VEL
LIN {X 0,Y 226.126,Z 400.494,A -85,B 0,C 180,E1 -20815.862,E2 -20815.862} C_VEL
LIN {X 0,Y 227.402,Z 364.424,A -85,B 0,C 180,E1 -20817.014,E2 -20817.014} C_VEL
LIN {X 0,Y 224.502,Z 347.056,A -85,B 0,C 180,E1 -20818.006,E2 -20818.006} C_VEL
LIN {X 0,Y 218.758,Z 332.595,A -85,B 0,C 180,E1 -20819.34,E2 -20819.34} C_VEL
LIN {X 0,Y 215.019,Z 324.041,A -85,B 0,C 180,E1 -20820.284,E2 -20820.284} C_VEL
LIN {X 0,Y 214.804,Z 323.14,A -85,B 0,C 180,E1 -20820.609,E2 -20820.609} C_VEL
LIN {X 0,Y 213.808,Z 318.763,A -85,B 0,C 180,E1 -20823.265,E2 -20823.265} C_VEL
LIN {X 0,Y 213.717,Z 318.677,A -85,B 0,C 180,E1 -20827.886,E2 -20827.886} C_VEL
LIN {X 0,Y 213.695,Z 318.644,A -85,B 0,C 180,E1 -20831.128,E2 -20831.128} C_VEL
LIN {X 0,Y 213.699,Z 318.661,A -85,B 0,C 180,E1 -20833.679,E2 -20833.679} C_VEL
LIN {X 0,Y 213.698,Z 318.679,A -85,B 0,C 180,E1 -20836.345,E2 -20836.345} C_VEL
LIN {X 0,Y 213.697,Z 318.627,A -85,B 0,C 180,E1 -20841.327,E2 -20841.327} C_VEL
LIN {X 0,Y 213.75,Z 318.67,A -85,B 0,C 180,E1 -20846.016,E2 -20846.016} C_VEL
LIN {X 0,Y 213.744,Z 318.656,A -85,B 0,C 180,E1 -20850.448,E2 -20850.448} C_VEL
LIN {X 0,Y 213.746,Z 318.672,A -85,B 0,C 180,E1 -20854.694,E2 -20854.694} C_VEL
LIN {X 0,Y 213.769,Z 318.652,A -85,B 0,C 180,E1 -20858.799,E2 -20858.799} C_VEL
LIN {X 0,Y 213.873,Z 318.654,A -85,B 0,C 180,E1 -20862.798,E2 -20862.798} C_VEL
LIN {X 0,Y 213.905,Z 318.631,A -85,B 0,C 180,E1 -20866.703,E2 -20866.703} C_VEL
LIN {X 0,Y 214.128,Z 318.624,A -85,B 0,C 180,E1 -20870.554,E2 -20870.554} C_VEL
LIN {X 0,Y 214.066,Z 318.61,A -85,B 0,C 180,E1 -20874.347,E2 -20874.347} C_VEL
LIN {X 0,Y 214.397,Z 318.585,A -85,B 0,C 180,E1 -20878.121,E2 -20878.121} C_VEL
LIN {X 0,Y 214.505,Z 318.58,A -85,B 0,C 180,E1 -20880,E2 -20880} C_VEL
LIN {X 0,Y 214.394,Z 318.586,A -85,B 0,C 180,E1 -20881.878,E2 -20881.878} C_VEL
LIN {X 0,Y 214.165,Z 318.613,A -85,B 0,C 180,E1 -20887.542,E2 -20887.542} C_VEL
LIN {X 0,Y 213.976,Z 318.635,A -85,B 0,C 180,E1 -20891.365,E2 -20891.365} C_VEL
LIN {X 0,Y 213.859,Z 318.644,A -85,B 0,C 180,E1 -20895.242,E2 -20895.242} C_VEL
LIN {X 0,Y 213.784,Z 318.666,A -85,B 0,C 180,E1 -20899.192,E2 -20899.192} C_VEL
LIN {X 0,Y 213.78,Z 318.652,A -85,B 0,C 180,E1 -20903.235,E2 -20903.235} C_VEL
LIN {X 0,Y 213.781,Z 318.664,A -85,B 0,C 180,E1 -20907.427,E2 -20907.427} C_VEL
LIN {X 0,Y 213.754,Z 318.668,A -85,B 0,C 180,E1 -20911.739,E2 -20911.739} C_VEL
LIN {X 0,Y 213.737,Z 318.648,A -85,B 0,C 180,E1 -20916.289,E2 -20916.289} C_VEL
LIN {X 0,Y 213.694,Z 318.645,A -85,B 0,C 180,E1 -20921.129,E2 -20921.129} C_VEL
LIN {X 0,Y 213.689,Z 318.678,A -85,B 0,C 180,E1 -20923.788,E2 -20923.788} C_VEL
LIN {X 0,Y 213.698,Z 318.662,A -85,B 0,C 180,E1 -20926.346,E2 -20926.346} C_VEL
LIN {X 0,Y 213.702,Z 318.672,A -85,B 0,C 180,E1 -20931.33,E2 -20931.33} C_VEL
LIN {X 0,Y 213.71,Z 318.676,A -85,B 0,C 180,E1 -20931.984,E2 -20931.984} C_VEL
LIN {X 0,Y 213.061,Z 318.755,A -85,B 0,C 180,E1 -20933.05,E2 -20933.05} C_VEL
LIN {X 0,Y 210.275,Z 319.172,A -85,B 0,C 180,E1 -20934.731,E2 -20934.731} C_VEL
LIN {X 0,Y 207.639,Z 320.441,A -85,B 0,C 180,E1 -20936.41,E2 -20936.41} C_VEL
LIN {X 0,Y 207.225,Z 321.798,A -85,B 0,C 180,E1 -20937.441,E2 -20937.441} C_VEL
LIN {X 0,Y 207.7,Z 323.83,A -85,B 0,C 180,E1 -20938.543,E2 -20938.543} C_VEL
LIN {X 0,Y 210.596,Z 330.318,A -85,B 0,C 180,E1 -20939.362,E2 -20939.362} C_VEL
LIN {X 0,Y 216.431,Z 343.944,A -85,B 0,C 180,E1 -20940.782,E2 -20940.782} C_VEL
LIN {X 0,Y 218.722,Z 350.416,A -85,B 0,C 180,E1 -20941.355,E2 -20941.355} C_VEL
LIN {X 0,Y 221.065,Z 365.835,A -85,B 0,C 180,E1 -20942.242,E2 -20942.242} C_VEL
LIN {X 0,Y 219.814,Z 401.028,A -85,B 0,C 180,E1 -20943.41,E2 -20943.41} C_VEL
LIN {X 0,Y 218.811,Z 412.714,A -85,B 0,C 180,E1 -20944.1,E2 -20944.1} C_VEL
LIN {X 0,Y 217.399,Z 423.727,A -85,B 0,C 180,E1 -20945.15,E2 -20945.15} C_VEL
LIN {X 0,Y 216.042,Z 432.39,A -85,B 0,C 180,E1 -20946.262,E2 -20946.262} C_VEL
LIN {X 0,Y 214.472,Z 440.668,A -85,B 0,C 180,E1 -20947.609,E2 -20947.609} C_VEL
LIN {X 0,Y 212.697,Z 448.505,A -85,B 0,C 180,E1 -20949.195,E2 -20949.195} C_VEL
LIN {X 0,Y 210.918,Z 455.832,A -85,B 0,C 180,E1 -20951.042,E2 -20951.042} C_VEL
LIN {X 0,Y 209.063,Z 463.264,A -85,B 0,C 180,E1 -20953.397,E2 -20953.397} C_VEL
LIN {X 0,Y 207.221,Z 470.042,A -85,B 0,C 180,E1 -20956.267,E2 -20956.267} C_VEL
LIN {X 0,Y 205.905,Z 475.191,A -85,B 0,C 180,E1 -20959.18,E2 -20959.18} C_VEL
LIN {X 0,Y 205.025,Z 478.969,A -85,B 0,C 180,E1 -20962.119,E2 -20962.119} C_VEL
LIN {X 0,Y 204.473,Z 481.614,A -85,B 0,C 180,E1 -20965.388,E2 -20965.388} C_VEL
LIN {X 0,Y 204.321,Z 482.71,A -85,B 0,C 180,E1 -20968.029,E2 -20968.029} C_VEL
LIN {X 0,Y 204.301,Z 483,A -85,B 0,C 180,E1 -20970,E2 -20970} C_VEL
LIN {X 0,Y 204.32,Z 482.701,A -85,B 0,C 180,E1 -20971.971,E2 -20971.971} C_VEL
LIN {X 0,Y 204.438,Z 481.649,A -85,B 0,C 180,E1 -20974.487,E2 -20974.487} C_VEL
LIN {X 0,Y 204.991,Z 478.905,A -85,B 0,C 180,E1 -20977.882,E2 -20977.882} C_VEL
LIN {X 0,Y 205.899,Z 475.108,A -85,B 0,C 180,E1 -20980.82,E2 -20980.82} C_VEL
LIN {X 0,Y 207.216,Z 469.934,A -85,B 0,C 180,E1 -20983.734,E2 -20983.734} C_VEL
LIN {X 0,Y 209.06,Z 463.107,A -85,B 0,C 180,E1 -20986.603,E2 -20986.603} C_VEL
LIN {X 0,Y 210.918,Z 455.646,A -85,B 0,C 180,E1 -20988.958,E2 -20988.958} C_VEL
LIN {X 0,Y 212.732,Z 448.285,A -85,B 0,C 180,E1 -20990.802,E2 -20990.802} C_VEL
LIN {X 0,Y 214.483,Z 440.398,A -85,B 0,C 180,E1 -20992.39,E2 -20992.39} C_VEL
LIN {X 0,Y 216.035,Z 432.058,A -85,B 0,C 180,E1 -20993.739,E2 -20993.739} C_VEL
LIN {X 0,Y 217.587,Z 422.046,A -85,B 0,C 180,E1 -20994.999,E2 -20994.999} C_VEL
LIN {X 0,Y 218.925,Z 410.67,A -85,B 0,C 180,E1 -20995.991,E2 -20995.991} C_VEL
LIN {X 0,Y 219.74,Z 400.836,A -85,B 0,C 180,E1 -20996.552,E2 -20996.552} C_VEL
LIN {X 0,Y 220.959,Z 365.314,A -85,B 0,C 180,E1 -20997.733,E2 -20997.733} C_VEL
LIN {X 0,Y 218.323,Z 349.04,A -85,B 0,C 180,E1 -20998.693,E2 -20998.693} C_VEL
LIN {X 0,Y 212.397,Z 334.305,A -85,B 0,C 180,E1 -21000.134,E2 -21000.134} C_VEL
LIN {X 0,Y 207.691,Z 323.901,A -85,B 0,C 180,E1 -21001.375,E2 -21001.375} C_VEL
LIN {X 0,Y 207.119,Z 321.167,A -85,B 0,C 180,E1 -21002.881,E2 -21002.881} C_VEL
LIN {X 0,Y 206.728,Z 319.62,A -85,B 0,C 180,E1 -21003.973,E2 -21003.973} C_VEL
LIN {X 0,Y 206.673,Z 319.546,A -85,B 0,C 180,E1 -21008.545,E2 -21008.545} C_VEL
LIN {X 0,Y 206.614,Z 319.533,A -85,B 0,C 180,E1 -21012.866,E2 -21012.866} C_VEL
LIN {X 0,Y 206.614,Z 319.553,A -85,B 0,C 180,E1 -21017.133,E2 -21017.133} C_VEL
LIN {X 0,Y 206.667,Z 319.501,A -85,B 0,C 180,E1 -21021.456,E2 -21021.456} C_VEL
LIN {X 0,Y 206.696,Z 319.539,A -85,B 0,C 180,E1 -21024.688,E2 -21024.688} C_VEL
LIN {X 0,Y 206.69,Z 319.537,A -85,B 0,C 180,E1 -21029.334,E2 -21029.334} C_VEL
LIN {X 0,Y 206.681,Z 319.552,A -85,B 0,C 180,E1 -21033.765,E2 -21033.765} C_VEL
LIN {X 0,Y 206.707,Z 319.528,A -85,B 0,C 180,E1 -21038.038,E2 -21038.038} C_VEL
LIN {X 0,Y 206.798,Z 319.539,A -85,B 0,C 180,E1 -21042.19,E2 -21042.19} C_VEL
LIN {X 0,Y 206.845,Z 319.508,A -85,B 0,C 180,E1 -21046.241,E2 -21046.241} C_VEL
LIN {X 0,Y 207.073,Z 319.503,A -85,B 0,C 180,E1 -21050.23,E2 -21050.23} C_VEL
LIN {X 0,Y 207.03,Z 319.487,A -85,B 0,C 180,E1 -21054.155,E2 -21054.155} C_VEL
LIN {X 0,Y 207.336,Z 319.463,A -85,B 0,C 180,E1 -21058.058,E2 -21058.058} C_VEL
LIN {X 0,Y 207.473,Z 319.455,A -85,B 0,C 180,E1 -21060,E2 -21060} C_VEL
LIN {X 0,Y 207.333,Z 319.464,A -85,B 0,C 180,E1 -21061.943,E2 -21061.943} C_VEL
LIN {X 0,Y 207.111,Z 319.493,A -85,B 0,C 180,E1 -21067.801,E2 -21067.801} C_VEL
LIN {X 0,Y 206.896,Z 319.513,A -85,B 0,C 180,E1 -21071.76,E2 -21071.76} C_VEL
LIN {X 0,Y 206.794,Z 319.526,A -85,B 0,C 180,E1 -21075.777,E2 -21075.777} C_VEL
LIN {X 0,Y 206.706,Z 319.543,A -85,B 0,C 180,E1 -21079.877,E2 -21079.877} C_VEL
LIN {X 0,Y 206.716,Z 319.538,A -85,B 0,C 180,E1 -21084.078,E2 -21084.078} C_VEL
LIN {X 0,Y 206.683,Z 319.542,A -85,B 0,C 180,E1 -21088.428,E2 -21088.428} C_VEL
LIN {X 0,Y 206.691,Z 319.552,A -85,B 0,C 180,E1 -21092.959,E2 -21092.959} C_VEL
LIN {X 0,Y 206.663,Z 319.508,A -85,B 0,C 180,E1 -21097.744,E2 -21097.744} C_VEL
LIN {X 0,Y 206.628,Z 319.527,A -85,B 0,C 180,E1 -21101.56,E2 -21101.56} C_VEL
LIN {X 0,Y 206.627,Z 319.554,A -85,B 0,C 180,E1 -21105.584,E2 -21105.584} C_VEL
LIN {X 0,Y 206.646,Z 319.524,A -85,B 0,C 180,E1 -21109.746,E2 -21109.746} C_VEL
LIN {X 0,Y 206.699,Z 319.531,A -85,B 0,C 180,E1 -21114.69,E2 -21114.69} C_VEL
LIN {X 0,Y 206.765,Z 319.685,A -85,B 0,C 180,E1 -21116.181,E2 -21116.181} C_VEL
LIN {X 0,Y 207.625,Z 323.715,A -85,B 0,C 180,E1 -21118.611,E2 -21118.611} C_VEL
LIN {X 0,Y 209.205,Z 327.331,A -85,B 0,C 180,E1 -21119.13,E2 -21119.13} C_VEL
LIN {X 0,Y 216.636,Z 344.483,A -85,B 0,C 180,E1 -21120.938,E2 -21120.938} C_VEL
LIN {X 0,Y 218.728,Z 350.8,A -85,B 0,C 180,E1 -21121.474,E2 -21121.474} C_VEL
